C07243=1098.667,-38.202,448.879,175.841,14.477,151.943
C07244=1098.673,-37.951,448.867,175.843,14.477,151.943
C07245=1098.679,-37.701,448.855,175.845,14.478,151.943
C07246=1098.684,-37.452,448.843,175.847,14.478,151.942
C07247=1098.691,-37.202,448.831,175.849,14.479,151.942
C07248=1098.697,-36.953,448.818,175.851,14.480,151.942
C07249=1098.702,-36.703,448.806,175.852,14.481,151.942
C07250=1098.708,-36.453,448.793,175.854,14.481,151.941
C07251=1098.714,-36.204,448.781,175.856,14.482,151.941
C07252=1098.720,-35.955,448.769,175.858,14.482,151.941
C07253=1098.726,-35.705,448.757,175.859,14.483,151.940
C07254=1098.732,-35.455,448.744,175.861,14.483,151.940
C07255=1098.738,-35.205,448.731,175.863,14.484,151.940
C07256=1098.743,-34.956,448.719,175.865,14.485,151.940
C07257=1098.749,-34.706,448.707,175.867,14.486,151.939
C07258=1098.755,-34.456,448.695,175.869,14.486,151.939
C07259=1098.761,-34.207,448.683,175.871,14.487,151.939
C07260=1098.767,-33.957,448.670,175.873,14.487,151.938
C07261=1098.773,-33.707,448.657,175.875,14.488,151.938
C07262=1098.778,-33.458,448.645,175.877,14.489,151.938
C07263=1098.784,-33.208,448.633,175.879,14.490,151.938
C07264=1098.790,-32.959,448.620,175.880,14.490,151.937
C07265=1098.797,-32.692,448.607,175.883,14.491,151.937
C07266=1098.803,-32.424,448.593,175.885,14.492,151.937
C07267=1098.809,-32.158,448.581,175.887,14.493,151.936
C07268=1098.815,-31.891,448.567,175.889,14.494,151.936
C07269=1098.821,-31.641,448.554,175.891,14.494,151.936
C07270=1098.827,-31.391,448.542,175.893,14.495,151.935
C07271=1098.832,-31.142,448.529,175.895,14.495,151.935
C07272=1098.838,-30.892,448.517,175.897,14.496,151.935
C07273=1098.845,-30.642,448.505,175.899,14.497,151.935
C07274=1098.851,-30.392,448.492,175.901,14.497,151.934
C07275=1098.857,-30.142,448.480,175.903,14.498,151.934
C07276=1098.862,-29.893,448.468,175.905,14.499,151.934
C07277=1098.868,-29.644,448.454,175.907,14.499,151.933
C07278=1098.874,-29.394,448.442,175.908,14.500,151.933
C07279=1098.880,-29.144,448.429,175.911,14.500,151.933
C07280=1098.886,-28.894,448.417,175.912,14.501,151.932
C07281=1098.891,-28.645,448.405,175.914,14.502,151.932
C07282=1098.897,-28.395,448.392,175.916,14.503,151.932
C07283=1098.903,-28.146,448.379,175.918,14.503,151.932
C07284=1098.909,-27.896,448.366,175.920,14.504,151.931
C07285=1098.916,-27.647,448.354,175.922,14.504,151.931
C07286=1098.921,-27.397,448.342,175.924,14.505,151.931
C07287=1098.928,-27.148,448.329,175.926,14.506,151.930
C07288=1098.933,-26.898,448.316,175.928,14.507,151.930
C07289=1098.939,-26.648,448.304,175.930,14.507,151.930
C07290=1098.945,-26.398,448.291,175.932,14.508,151.930
C07291=1098.950,-26.149,448.278,175.934,14.509,151.929
C07292=1098.956,-25.900,448.265,175.936,14.509,151.929
C07293=1098.962,-25.650,448.252,175.937,14.510,151.929
C07294=1098.968,-25.400,448.240,175.939,14.511,151.928
C07295=1098.974,-25.150,448.227,175.942,14.511,151.928
C07296=1098.979,-24.902,448.214,175.943,14.512,151.928
C07297=1098.985,-24.652,448.202,175.945,14.513,151.928
C07298=1098.991,-24.402,448.189,175.947,14.513,151.927
C07299=1098.997,-24.152,448.176,175.949,14.514,151.927
C07300=1099.003,-23.902,448.163,175.951,14.515,151.927
C07301=1099.008,-23.652,448.150,175.953,14.515,151.926
C07302=1099.014,-23.404,448.138,175.956,14.517,151.926
C07303=1099.020,-23.154,448.125,175.958,14.517,151.926
C07304=1099.026,-22.904,448.112,175.960,14.518,151.926
C07305=1099.032,-22.655,448.099,175.961,14.519,151.925
C07306=1099.038,-22.405,448.087,175.964,14.519,151.925
C07307=1099.044,-22.155,448.074,175.965,14.520,151.925
C07308=1099.049,-21.906,448.061,175.967,14.521,151.924
C07309=1099.055,-21.656,448.048,175.969,14.521,151.924
C07310=1099.061,-21.406,448.035,175.971,14.522,151.924
C07311=1099.067,-21.157,448.022,175.973,14.522,151.923
C07312=1099.073,-20.907,448.010,175.975,14.523,151.923
C07313=1099.079,-20.658,447.996,175.977,14.524,151.923
C07314=1099.085,-20.408,447.984,175.979,14.525,151.923
C07315=1099.090,-20.158,447.971,175.981,14.525,151.922
C07316=1099.096,-19.909,447.957,175.983,14.526,151.922
C07317=1099.102,-19.659,447.945,175.985,14.527,151.922
C07318=1099.108,-19.410,447.932,175.987,14.527,151.921
C07319=1099.114,-19.160,447.919,175.989,14.528,151.921
C07320=1099.119,-18.911,447.905,175.991,14.528,151.921
C07321=1099.125,-18.661,447.893,175.993,14.529,151.920
C07322=1099.131,-18.412,447.880,175.995,14.530,151.920
C07323=1099.137,-18.162,447.867,175.997,14.531,151.920
C07324=1099.143,-17.912,447.855,175.999,14.531,151.919
C07325=1099.149,-17.662,447.841,176.001,14.532,151.919
C07326=1099.154,-17.412,447.828,176.003,14.533,151.919
C07327=1099.161,-17.163,447.815,176.005,14.534,151.919
C07328=1099.167,-16.914,447.802,176.007,14.534,151.918
C07329=1099.173,-16.646,447.789,176.009,14.535,151.918
C07330=1099.179,-16.378,447.774,176.011,14.536,151.918
C07331=1099.185,-16.110,447.760,176.014,14.536,151.917
C07332=1099.192,-15.842,447.746,176.016,14.537,151.917
C07333=1099.198,-15.593,447.733,176.018,14.538,151.917
C07334=1099.203,-15.343,447.720,176.020,14.538,151.916
C07335=1099.209,-15.094,447.706,176.022,14.539,151.916
C07336=1099.215,-14.844,447.694,176.024,14.540,151.916
C07337=1099.221,-14.594,447.680,176.025,14.541,151.916
C07338=1099.227,-14.344,447.667,176.028,14.541,151.915
C07339=1099.233,-14.095,447.654,176.030,14.542,151.915
C07340=1099.238,-13.845,447.640,176.031,14.542,151.915
C07341=1099.244,-13.595,447.628,176.034,14.544,151.914
C07342=1099.249,-13.347,447.614,176.036,14.544,151.914
C07343=1099.255,-13.097,447.602,176.038,14.545,151.914
C07344=1099.261,-12.847,447.588,176.040,14.546,151.913
C07345=1099.267,-12.598,447.574,176.042,14.546,151.913
C07346=1099.273,-12.348,447.562,176.044,14.547,151.913
C07347=1099.278,-12.098,447.548,176.046,14.547,151.912
C07348=1099.284,-11.849,447.535,176.048,14.548,151.912
C07349=1099.290,-11.599,447.522,176.050,14.549,151.912
C07350=1099.296,-11.350,447.508,176.052,14.549,151.912
C07351=1099.302,-11.100,447.495,176.054,14.550,151.911
C07352=1099.307,-10.850,447.482,176.056,14.551,151.911
C07353=1099.313,-10.601,447.469,176.058,14.552,151.911
C07354=1099.319,-10.351,447.455,176.060,14.552,151.910
C07355=1099.325,-10.101,447.442,176.062,14.553,151.910
C07356=1099.331,-9.852,447.429,176.064,14.554,151.910
C07357=1099.336,-9.603,447.415,176.066,14.554,151.909
C07358=1099.343,-9.353,447.402,176.068,14.555,151.909
C07359=1099.348,-9.103,447.389,176.070,14.556,151.909
C07360=1099.354,-8.854,447.375,176.072,14.556,151.908
C07361=1099.359,-8.604,447.362,176.074,14.557,151.908
C07362=1099.366,-8.355,447.348,176.077,14.558,151.908
C07363=1099.371,-8.105,447.335,176.079,14.559,151.908
C07364=1099.377,-7.856,447.322,176.081,14.559,151.907
C07365=1099.383,-7.606,447.308,176.083,14.560,151.907
C07366=1099.389,-7.357,447.295,176.085,14.561,151.907
C07367=1099.395,-7.106,447.282,176.087,14.561,151.906
C07368=1099.401,-6.857,447.268,176.089,14.562,151.906
C07369=1099.407,-6.607,447.255,176.091,14.563,151.906
C07370=1099.412,-6.358,447.241,176.093,14.563,151.905
C07371=1099.419,-6.109,447.228,176.095,14.564,151.905
C07372=1099.424,-5.859,447.214,176.097,14.565,151.905
C07373=1099.430,-5.609,447.201,176.100,14.565,151.904
C07374=1099.436,-5.360,447.187,176.101,14.566,151.904
C07375=1099.442,-5.110,447.174,176.104,14.566,151.904
C07376=1099.447,-4.861,447.160,176.105,14.567,151.903
C07377=1099.453,-4.611,447.147,176.107,14.568,151.903
C07378=1099.459,-4.362,447.133,176.110,14.568,151.903
C07379=1099.466,-4.112,447.119,176.111,14.569,151.902
C07380=1099.471,-3.862,447.106,176.114,14.570,151.902
C07381=1099.476,-3.612,447.092,176.116,14.571,151.902
C07382=1099.483,-3.363,447.079,176.118,14.571,151.901
C07383=1099.488,-3.113,447.065,176.120,14.572,151.901
C07384=1099.494,-2.864,447.052,176.122,14.572,151.901
C07385=1099.500,-2.614,447.038,176.124,14.573,151.901
C07386=1099.505,-2.365,447.024,176.126,14.574,151.900
C07387=1099.511,-2.115,447.010,176.128,14.574,151.900
C07388=1099.517,-1.866,446.997,176.131,14.576,151.900
C07389=1099.522,-1.616,446.983,176.133,14.576,151.899
C07390=1099.528,-1.367,446.969,176.135,14.577,151.899
C07391=1099.534,-1.118,446.956,176.137,14.577,151.899
C07392=1099.540,-0.867,446.942,176.139,14.578,151.898
C07393=1099.546,-0.597,446.927,176.141,14.578,151.898
C07394=1099.552,-0.328,446.912,176.143,14.580,151.898
C07395=1099.559,-0.059,446.898,176.146,14.580,151.897
C07396=1099.564,0.211,446.883,176.147,14.581,151.897
C07397=1099.571,0.461,446.869,176.150,14.582,151.897
C07398=1099.576,0.710,446.855,176.152,14.583,151.896
C07399=1099.581,0.960,446.842,176.154,14.583,151.896
C07400=1099.587,1.209,446.828,176.156,14.584,151.896
C07401=1099.593,1.459,446.814,176.158,14.584,151.895
C07402=1099.599,1.708,446.800,176.160,14.585,151.895
C07403=1099.604,1.957,446.786,176.162,14.585,151.895
C07404=1099.610,2.207,446.772,176.165,14.587,151.894
C07405=1099.616,2.457,446.758,176.167,14.588,151.894
C07406=1099.622,2.706,446.745,176.169,14.588,151.894
C07407=1099.628,2.956,446.731,176.171,14.589,151.893
C07408=1099.633,3.205,446.717,176.173,14.589,151.893
C07409=1099.639,3.455,446.703,176.175,14.590,151.893
C07410=1099.644,3.705,446.689,176.178,14.591,151.892
C07411=1099.651,3.955,446.676,176.180,14.591,151.892
C07412=1099.657,4.204,446.661,176.182,14.592,151.892
C07413=1099.662,4.453,446.647,176.184,14.592,151.891
C07414=1099.668,4.703,446.633,176.186,14.593,151.891
C07415=1099.673,4.952,446.619,176.188,14.594,151.891
C07416=1099.679,5.201,446.606,176.190,14.594,151.890
C07417=1099.685,5.452,446.592,176.192,14.596,151.890
C07418=1099.691,5.701,446.577,176.195,14.596,151.890
C07419=1099.697,5.950,446.563,176.196,14.597,151.889
C07420=1099.702,6.200,446.550,176.199,14.597,151.889
C07421=1099.708,6.450,446.535,176.201,14.598,151.889
C07422=1099.714,6.699,446.522,176.203,14.598,151.888
C07423=1099.720,6.948,446.507,176.205,14.599,151.888
C07424=1099.726,7.198,446.494,176.208,14.600,151.888
C07425=1099.731,7.448,446.480,176.209,14.601,151.887
C07426=1099.737,7.698,446.466,176.212,14.601,151.887
C07427=1099.743,7.947,446.451,176.214,14.602,151.887
C07428=1099.749,8.196,446.438,176.216,14.602,151.886
C07429=1099.755,8.446,446.424,176.218,14.603,151.886
C07430=1099.761,8.696,446.410,176.221,14.604,151.886
C07431=1099.767,8.945,446.395,176.222,14.604,151.885
C07432=1099.772,9.194,446.381,176.225,14.605,151.885
C07433=1099.778,9.444,446.367,176.226,14.605,151.885
C07434=1099.784,9.694,446.352,176.229,14.606,151.884
C07435=1099.789,9.943,446.338,176.231,14.607,151.884
C07436=1099.795,10.193,446.325,176.234,14.607,151.884
C07437=1099.802,10.442,446.310,176.235,14.608,151.883
C07438=1099.807,10.692,446.296,176.238,14.608,151.883
C07439=1099.813,10.941,446.283,176.239,14.609,151.883
C07440=1099.819,11.190,446.268,176.242,14.610,151.882
C07441=1099.825,11.441,446.254,176.244,14.611,151.882
C07442=1099.830,11.690,446.240,176.246,14.611,151.881
C07443=1099.836,11.939,446.225,176.248,14.612,151.881
C07444=1099.842,12.189,446.211,176.251,14.612,151.881
C07445=1099.848,12.438,446.196,176.253,14.613,151.880
C07446=1099.853,12.688,446.183,176.255,14.614,151.880
C07447=1099.859,12.938,446.168,176.258,14.614,151.880
C07448=1099.865,13.187,446.154,176.259,14.615,151.879
C07449=1099.871,13.437,446.140,176.262,14.615,151.879
C07450=1099.878,13.686,446.126,176.264,14.616,151.879
C07451=1099.883,13.936,446.112,176.266,14.617,151.878
C07452=1099.889,14.185,446.097,176.269,14.617,151.878
C07453=1099.895,14.435,446.083,176.271,14.618,151.878
C07454=1099.901,14.684,446.068,176.273,14.618,151.877
C07455=1099.906,14.934,446.054,176.275,14.619,151.877
C07456=1099.912,15.183,446.039,176.277,14.619,151.876
C07457=1099.918,15.455,446.024,176.280,14.620,151.876
C07458=1099.924,15.726,446.008,176.282,14.621,151.876
C07459=1099.931,15.998,445.992,176.285,14.622,151.875
C07460=1099.938,16.269,445.977,176.287,14.622,151.875
C07461=1099.942,16.519,445.962,176.289,14.623,151.875
C07462=1099.948,16.768,445.948,176.291,14.623,151.874
C07463=1099.954,17.018,445.933,176.294,14.624,151.874
C07464=1099.960,17.267,445.919,176.296,14.625,151.874
C07465=1099.965,17.517,445.905,176.298,14.625,151.873
C07466=1099.972,17.767,445.890,176.300,14.626,151.873
C07467=1099.977,18.016,445.876,176.303,14.627,151.872
C07468=1099.984,18.266,445.861,176.305,14.627,151.872
C07469=1099.989,18.515,445.846,176.307,14.628,151.872
C07470=1099.994,18.765,445.832,176.309,14.628,151.871
C07471=1100.001,19.014,445.817,176.311,14.629,151.871
C07472=1100.006,19.264,445.803,176.314,14.630,151.871
C07473=1100.012,19.513,445.789,176.316,14.630,151.870
C07474=1100.018,19.762,445.774,176.318,14.631,151.870
C07475=1100.023,20.012,445.759,176.320,14.632,151.869
C07476=1100.029,20.262,445.744,176.322,14.632,151.869
C07477=1100.035,20.511,445.730,176.325,14.633,151.869
C07478=1100.041,20.761,445.716,176.327,14.634,151.868
C07479=1100.047,21.010,445.701,176.329,14.634,151.868
C07480=1100.052,21.259,445.686,176.331,14.635,151.868
C07481=1100.058,21.510,445.672,176.334,14.636,151.867
C07482=1100.064,21.759,445.657,176.336,14.636,151.867
C07483=1100.070,22.008,445.642,176.338,14.637,151.867
C07484=1100.075,22.258,445.628,176.340,14.637,151.866
C07485=1100.081,22.507,445.613,176.342,14.638,151.866
C07486=1100.087,22.757,445.598,176.345,14.639,151.865
C07487=1100.092,23.006,445.583,176.347,14.639,151.865
C07488=1100.098,23.256,445.569,176.350,14.639,151.865
C07489=1100.104,23.505,445.554,176.351,14.640,151.864
C07490=1100.110,23.754,445.540,176.354,14.641,151.864
C07491=1100.116,24.004,445.524,176.357,14.641,151.863
C07492=1100.121,24.254,445.510,176.358,14.642,151.863
C07493=1100.127,24.503,445.495,176.361,14.642,151.863
C07494=1100.132,24.753,445.480,176.363,14.643,151.862
C07495=1100.138,25.002,445.465,176.365,14.644,151.862
C07496=1100.144,25.252,445.451,176.368,14.644,151.862
C07497=1100.149,25.501,445.436,176.370,14.645,151.861
C07498=1100.156,25.751,445.421,176.372,14.645,151.861
C07499=1100.162,26.000,445.407,176.375,14.646,151.861
C07500=1100.167,26.250,445.391,176.377,14.647,151.860
C07501=1100.173,26.499,445.376,176.379,14.647,151.860
C07502=1100.179,26.748,445.361,176.381,14.647,151.859
C07503=1100.184,26.998,445.347,176.384,14.649,151.859
C07504=1100.190,27.248,445.332,176.386,14.649,151.859
C07505=1100.196,27.497,445.317,176.388,14.649,151.858
C07506=1100.202,27.747,445.302,176.390,14.650,151.858
C07507=1100.208,27.996,445.287,176.393,14.650,151.857
C07508=1100.214,28.246,445.272,176.395,14.651,151.857
C07509=1100.219,28.495,445.257,176.398,14.652,151.857
C07510=1100.225,28.744,445.242,176.400,14.652,151.856
C07511=1100.231,28.994,445.227,176.403,14.653,151.856
C07512=1100.237,29.243,445.212,176.405,14.654,151.856
C07513=1100.242,29.493,445.198,176.407,14.654,151.855
C07514=1100.248,29.743,445.183,176.409,14.654,151.855
C07515=1100.253,29.992,445.168,176.412,14.655,151.854
C07516=1100.259,30.242,445.153,176.414,14.655,151.854
C07517=1100.265,30.491,445.137,176.416,14.656,151.854
C07518=1100.271,30.741,445.123,176.418,14.656,151.853
C07519=1100.276,30.990,445.107,176.421,14.657,151.853
C07520=1100.282,31.240,445.092,176.423,14.658,151.852
C07521=1100.288,31.512,445.075,176.425,14.658,151.852
C07522=1100.295,31.785,445.059,176.428,14.659,151.851
C07523=1100.301,32.058,445.043,176.431,14.659,151.851
C07524=1100.307,32.331,445.026,176.434,14.660,151.851
C07525=1100.313,32.581,445.011,176.436,14.660,151.850
C07526=1100.318,32.830,444.996,176.438,14.661,151.850
C07527=1100.325,33.080,444.981,176.440,14.662,151.849
C07528=1100.330,33.329,444.966,176.443,14.663,151.849
C07529=1100.336,33.579,444.951,176.445,14.663,151.849
C07530=1100.341,33.827,444.935,176.447,14.663,151.848
C07531=1100.348,34.077,444.920,176.450,14.664,151.848
C07532=1100.353,34.327,444.905,176.452,14.664,151.847
C07533=1100.358,34.576,444.889,176.455,14.665,151.847
C07534=1100.365,34.826,444.874,176.456,14.665,151.847
C07535=1100.370,35.075,444.859,176.459,14.666,151.846
C07536=1100.376,35.325,444.844,176.462,14.667,151.846
C07537=1100.382,35.575,444.829,176.464,14.667,151.845
C07538=1100.388,35.823,444.813,176.466,14.667,151.845
C07539=1100.394,36.073,444.798,176.469,14.668,151.844
C07540=1100.399,36.322,444.783,176.471,14.669,151.844
C07541=1100.405,36.572,444.768,176.473,14.669,151.844
C07542=1100.411,36.822,444.752,176.475,14.669,151.843
C07543=1100.417,37.071,444.738,176.478,14.670,151.843
C07544=1100.422,37.320,444.721,176.481,14.670,151.842
C07545=1100.428,37.570,444.706,176.483,14.671,151.842
C07546=1100.434,37.819,444.691,176.486,14.672,151.841
C07547=1100.440,38.069,444.676,176.488,14.672,151.841
C07548=1100.445,38.318,444.660,176.490,14.672,151.841
C07549=1100.451,38.568,444.645,176.492,14.673,151.840
C07550=1100.457,38.818,444.629,176.495,14.674,151.840
C07551=1100.462,39.067,444.614,176.497,14.674,151.840
C07552=1100.468,39.316,444.598,176.499,14.675,151.839
C07553=1100.474,39.565,444.583,176.502,14.676,151.839
C07554=1100.479,39.815,444.568,176.504,14.676,151.838
C07555=1100.485,40.065,444.552,176.507,14.676,151.838
C07556=1100.490,40.314,444.536,176.509,14.676,151.837
C07557=1100.497,40.563,444.521,176.512,14.677,151.837
C07558=1100.502,40.813,444.506,176.514,14.678,151.837
C07559=1100.508,41.062,444.490,176.516,14.678,151.836
C07560=1100.513,41.312,444.474,176.519,14.679,151.836
C07561=1100.519,41.562,444.459,176.521,14.679,151.835
C07562=1100.525,41.810,444.444,176.524,14.680,151.835
C07563=1100.531,42.060,444.428,176.526,14.680,151.834
C07564=1100.536,42.310,444.413,176.529,14.681,151.834
C07565=1100.542,42.559,444.397,176.531,14.681,151.834
C07566=1100.548,42.809,444.382,176.533,14.681,151.833
C07567=1100.554,43.058,444.365,176.536,14.682,151.833
C07568=1100.559,43.307,444.350,176.538,14.683,151.832
C07569=1100.565,43.557,444.335,176.541,14.683,151.832
C07570=1100.571,43.806,444.318,176.544,14.684,151.831
C07571=1100.576,44.056,444.303,176.546,14.684,151.831
C07572=1100.582,44.305,444.287,176.548,14.684,151.830
C07573=1100.587,44.555,444.271,176.550,14.684,151.830
C07574=1100.592,44.804,444.256,176.553,14.685,151.830
C07575=1100.599,45.053,444.241,176.555,14.686,151.829
C07576=1100.605,45.303,444.225,176.558,14.686,151.829
C07577=1100.610,45.552,444.209,176.561,14.687,151.828
C07578=1100.616,45.802,444.194,176.563,14.687,151.828
C07579=1100.622,46.051,444.177,176.565,14.688,151.827
C07580=1100.627,46.301,444.162,176.568,14.689,151.827
C07581=1100.633,46.550,444.146,176.570,14.689,151.827
C07582=1100.638,46.800,444.130,176.572,14.689,151.826
C07583=1100.644,47.049,444.114,176.575,14.690,151.826
C07584=1100.649,47.298,444.099,176.577,14.690,151.825
C07585=1100.656,47.572,444.081,176.580,14.691,151.825
C07586=1100.662,47.845,444.064,176.583,14.691,151.824
C07587=1100.668,48.117,444.047,176.586,14.692,151.824
C07588=1100.674,48.391,444.029,176.588,14.692,151.823
C07589=1100.680,48.640,444.013,176.591,14.692,151.823
C07590=1100.685,48.889,443.997,176.594,14.693,151.822
C07591=1100.691,49.139,443.982,176.596,14.694,151.822
C07592=1100.697,49.388,443.965,176.598,14.694,151.822
C07593=1100.702,49.637,443.950,176.601,14.695,151.821
C07594=1100.708,49.887,443.934,176.603,14.695,151.821
C07595=1100.714,50.136,443.918,176.605,14.695,151.820
C07596=1100.720,50.386,443.902,176.609,14.696,151.820
C07597=1100.726,50.636,443.886,176.611,14.696,151.819
C07598=1100.731,50.884,443.870,176.613,14.697,151.819
C07599=1100.737,51.134,443.854,176.616,14.698,151.818
C07600=1100.743,51.383,443.838,176.618,14.698,151.818
C07601=1100.748,51.633,443.821,176.621,14.698,151.817
C07602=1100.753,51.883,443.806,176.624,14.699,151.817
C07603=1100.759,52.132,443.790,176.626,14.699,151.817
C07604=1100.765,52.381,443.774,176.628,14.699,151.816
C07605=1100.770,52.631,443.758,176.631,14.700,151.815
C07606=1100.776,52.880,443.742,176.633,14.700,151.815
C07607=1100.782,53.130,443.726,176.636,14.700,151.815
C07608=1100.788,53.378,443.710,176.638,14.701,151.814
C07609=1100.793,53.628,443.694,176.641,14.701,151.814
C07610=1100.799,53.878,443.678,176.643,14.702,151.813
C07611=1100.805,54.127,443.662,176.645,14.702,151.813
C07612=1100.811,54.376,443.645,176.648,14.703,151.812
C07613=1100.816,54.627,443.629,176.651,14.703,151.812
C07614=1100.822,54.876,443.613,176.653,14.703,151.811
C07615=1100.827,55.125,443.597,176.656,14.704,151.811
C07616=1100.833,55.374,443.581,176.659,14.704,151.810
C07617=1100.839,55.623,443.565,176.661,14.704,151.810
C07618=1100.845,55.873,443.548,176.664,14.705,151.809
C07619=1100.851,56.123,443.533,176.666,14.705,151.809
C07620=1100.856,56.372,443.516,176.668,14.705,151.808
C07621=1100.862,56.622,443.500,176.671,14.706,151.808
C07622=1100.868,56.871,443.483,176.674,14.706,151.807
C07623=1100.874,57.120,443.467,176.676,14.706,151.807
C07624=1100.879,57.369,443.451,176.679,14.707,151.806
C07625=1100.885,57.618,443.435,176.681,14.707,151.806
C07626=1100.891,57.868,443.419,176.684,14.707,151.806
C07627=1100.896,58.118,443.403,176.687,14.708,151.805
C07628=1100.902,58.367,443.386,176.689,14.708,151.805
C07629=1100.908,58.617,443.370,176.692,14.708,151.804
C07630=1100.914,58.866,443.354,176.695,14.709,151.804
C07631=1100.920,59.115,443.338,176.697,14.709,151.803
C07632=1100.925,59.365,443.321,176.700,14.710,151.803
C07633=1100.931,59.614,443.305,176.702,14.710,151.802
C07634=1100.937,59.864,443.288,176.705,14.710,151.802
C07635=1100.943,60.113,443.272,176.708,14.711,151.801
C07636=1100.949,60.362,443.256,176.710,14.711,151.801
C07637=1100.954,60.612,443.239,176.712,14.711,151.800
C07638=1100.960,60.861,443.223,176.716,14.712,151.799
C07639=1100.966,61.111,443.206,176.718,14.712,151.799
C07640=1100.972,61.360,443.190,176.720,14.712,151.798
C07641=1100.977,61.610,443.173,176.723,14.713,151.798
C07642=1100.983,61.859,443.157,176.726,14.713,151.797
C07643=1100.989,62.109,443.141,176.728,14.713,151.797
C07644=1100.995,62.357,443.124,176.731,14.714,151.796
C07645=1101.001,62.607,443.107,176.734,14.714,151.796
C07646=1101.006,62.856,443.091,176.736,14.714,151.795
C07647=1101.012,63.106,443.074,176.739,14.715,151.795
C07648=1101.018,63.355,443.058,176.741,14.715,151.794
C07649=1101.025,63.627,443.040,176.745,14.715,151.794
C07650=1101.030,63.901,443.022,176.747,14.715,151.793
C07651=1101.037,64.174,443.004,176.750,14.716,151.793
C07652=1101.043,64.446,442.986,176.753,14.716,151.792
C07653=1101.049,64.695,442.970,176.756,14.716,151.792
C07654=1101.055,64.945,442.953,176.758,14.717,151.791
C07655=1101.061,65.194,442.936,176.761,14.716,151.791
C07656=1101.066,65.443,442.919,176.764,14.717,151.790
C07657=1101.072,65.693,442.903,176.766,14.717,151.790
C07658=1101.078,65.942,442.886,176.769,14.717,151.789
C07659=1101.083,66.192,442.870,176.772,14.718,151.789
C07660=1101.089,66.441,442.853,176.774,14.718,151.788
C07661=1101.095,66.690,442.836,176.776,14.718,151.788
C07662=1101.101,66.939,442.819,176.780,14.719,151.787
C07663=1101.106,67.189,442.803,176.782,14.719,151.786
C07664=1101.112,67.438,442.786,176.785,14.720,151.786
C07665=1101.117,67.688,442.769,176.788,14.719,151.785
C07666=1101.124,67.937,442.752,176.790,14.720,151.785
C07667=1101.129,68.187,442.735,176.793,14.720,151.784
C07668=1101.135,68.436,442.719,176.796,14.720,151.784
C07669=1101.141,68.686,442.701,176.798,14.720,151.783
C07670=1101.146,68.935,442.685,176.801,14.721,151.783
C07671=1101.152,69.185,442.668,176.804,14.721,151.782
C07672=1101.158,69.433,442.651,176.806,14.722,151.782
C07673=1101.163,69.683,442.635,176.809,14.722,151.781
C07674=1101.169,69.932,442.618,176.812,14.721,151.781
C07675=1101.174,70.182,442.601,176.814,14.722,151.780
C07676=1101.181,70.431,442.584,176.817,14.722,151.780
C07677=1101.186,70.680,442.568,176.819,14.722,151.779
C07678=1101.191,70.929,442.550,176.822,14.723,151.779
C07679=1101.197,71.179,442.534,176.825,14.723,151.778
C07680=1101.203,71.429,442.517,176.828,14.724,151.777
C07681=1101.209,71.678,442.500,176.830,14.724,151.777
C07682=1101.215,71.927,442.483,176.833,14.724,151.776
C07683=1101.220,72.176,442.465,176.836,14.724,151.776
C07684=1101.226,72.426,442.449,176.838,14.725,151.775
C07685=1101.231,72.675,442.432,176.841,14.724,151.775
C07686=1101.237,72.925,442.414,176.844,14.725,151.774
C07687=1101.243,73.174,442.398,176.847,14.725,151.774
C07688=1101.248,73.423,442.381,176.850,14.726,151.773
C07689=1101.255,73.673,442.364,176.852,14.726,151.773
C07690=1101.260,73.922,442.346,176.855,14.725,151.772
C07691=1101.265,74.172,442.330,176.858,14.726,151.771
C07692=1101.272,74.420,442.313,176.860,14.726,151.771
C07693=1101.277,74.670,442.296,176.863,14.726,151.770
C07694=1101.282,74.919,442.278,176.866,14.727,151.770
C07695=1101.288,75.169,442.261,176.868,14.727,151.769
C07696=1101.295,75.418,442.244,176.872,14.727,151.769
C07697=1101.300,75.668,442.227,176.874,14.727,151.768
C07698=1101.305,75.917,442.210,176.876,14.727,151.768
C07699=1101.311,76.166,442.193,176.880,14.728,151.767
C07700=1101.317,76.415,442.176,176.882,14.728,151.766
C07701=1101.322,76.665,442.159,176.885,14.728,151.766
C07702=1101.329,76.914,442.142,176.888,14.728,151.765
C07703=1101.334,77.163,442.124,176.890,14.728,151.765
C07704=1101.340,77.413,442.107,176.893,14.729,151.764
C07705=1101.345,77.662,442.090,176.896,14.729,151.764
C07706=1101.351,77.911,442.073,176.898,14.729,151.763
C07707=1101.357,78.161,442.055,176.902,14.729,151.762
C07708=1101.363,78.410,442.038,176.904,14.729,151.762
C07709=1101.368,78.660,442.021,176.907,14.730,151.761
C07710=1101.373,78.909,442.003,176.910,14.729,151.761
C07711=1101.380,79.158,441.986,176.912,14.729,151.760
C07712=1101.385,79.408,441.969,176.916,14.730,151.760
C07713=1101.391,79.680,441.950,176.918,14.730,151.759
C07714=1101.397,79.953,441.931,176.922,14.730,151.758
C07715=1101.404,80.226,441.911,176.925,14.731,151.758
C07716=1101.410,80.499,441.893,176.927,14.731,151.757
C07717=1101.416,80.747,441.876,176.931,14.731,151.757
C07718=1101.421,80.997,441.859,176.933,14.731,151.756
C07719=1101.427,81.246,441.841,176.936,14.731,151.755
C07720=1101.432,81.495,441.824,176.939,14.731,151.755
C07721=1101.438,81.745,441.806,176.941,14.731,151.754
C07722=1101.444,81.995,441.789,176.945,14.732,151.754
C07723=1101.449,82.244,441.771,176.947,14.732,151.753
C07724=1101.455,82.493,441.754,176.950,14.732,151.752
C07725=1101.461,82.742,441.736,176.953,14.732,151.752
C07726=1101.466,82.991,441.718,176.955,14.732,151.751
C07727=1101.472,83.241,441.701,176.959,14.732,151.751
C07728=1101.477,83.490,441.684,176.961,14.732,151.750
C07729=1101.483,83.740,441.666,176.965,14.733,151.750
C07730=1101.489,83.989,441.648,176.967,14.733,151.749
C07731=1101.494,84.238,441.631,176.970,14.733,151.748
C07732=1101.500,84.488,441.613,176.973,14.733,151.748
C07733=1101.506,84.737,441.597,176.975,14.733,151.747
C07734=1101.512,84.986,441.579,176.979,14.733,151.747
C07735=1101.517,85.235,441.561,176.981,14.733,151.746
C07736=1101.523,85.485,441.543,176.984,14.733,151.745
C07737=1101.529,85.734,441.526,176.987,14.734,151.745
C07738=1101.534,85.983,441.508,176.989,14.734,151.744
C07739=1101.541,86.233,441.490,176.993,14.734,151.744
C07740=1101.546,86.482,441.473,176.995,14.734,151.743
C07741=1101.552,86.731,441.455,176.998,14.733,151.742
C07742=1101.558,86.980,441.437,177.001,14.734,151.742
C07743=1101.563,87.230,441.420,177.004,14.734,151.741
C07744=1101.569,87.479,441.402,177.007,14.734,151.741
C07745=1101.575,87.728,441.384,177.010,14.734,151.740
C07746=1101.580,87.978,441.366,177.012,14.734,151.739
C07747=1101.586,88.227,441.348,177.016,14.734,151.739
C07748=1101.591,88.476,441.331,177.018,14.734,151.738
C07749=1101.597,88.725,441.313,177.021,14.735,151.737
C07750=1101.603,88.975,441.295,177.024,14.734,151.737
C07751=1101.608,89.224,441.278,177.026,14.734,151.736
C07752=1101.615,89.474,441.260,177.030,14.734,151.736
C07753=1101.620,89.723,441.242,177.033,14.734,151.735
C07754=1101.626,89.972,441.224,177.036,14.735,151.734
C07755=1101.632,90.222,441.207,177.038,14.735,151.734
C07756=1101.637,90.471,441.189,177.042,14.735,151.733
C07757=1101.643,90.721,441.171,177.044,14.735,151.732
C07758=1101.649,90.970,441.153,177.047,14.735,151.732
C07759=1101.655,91.218,441.135,177.050,14.735,151.731
C07760=1101.660,91.468,441.117,177.053,14.734,151.731
C07761=1101.666,91.717,441.099,177.056,14.735,151.730
C07762=1101.672,91.967,441.081,177.059,14.735,151.729
C07763=1101.677,92.216,441.064,177.061,14.735,151.729
C07764=1101.682,92.465,441.045,177.065,14.735,151.728
C07765=1101.688,92.715,441.027,177.067,14.735,151.727
C07766=1101.694,92.963,441.009,177.071,14.735,151.727
C07767=1101.700,93.213,440.991,177.073,14.735,151.726
C07768=1101.706,93.462,440.974,177.077,14.735,151.726
C07769=1101.710,93.712,440.956,177.079,14.735,151.725
C07770=1101.717,93.961,440.938,177.082,14.735,151.724
C07771=1101.722,94.210,440.919,177.085,14.736,151.724
C07772=1101.728,94.460,440.901,177.088,14.735,151.723
C07773=1101.733,94.709,440.883,177.091,14.736,151.722
C07774=1101.739,94.959,440.865,177.094,14.735,151.722
C07775=1101.745,95.207,440.847,177.097,14.735,151.721
C07776=1101.750,95.456,440.829,177.100,14.735,151.721
C07777=1101.757,95.730,440.809,177.103,14.735,151.720
C07778=1101.763,96.002,440.789,177.106,14.735,151.719
C07779=1101.769,96.275,440.769,177.109,14.735,151.718
C07780=1101.775,96.547,440.749,177.113,14.735,151.718
C07781=1101.781,96.797,440.732,177.116,14.735,151.717
C07782=1101.787,97.046,440.713,177.118,14.735,151.716
C07783=1101.792,97.295,440.695,177.122,14.735,151.716
C07784=1101.798,97.545,440.677,177.124,14.735,151.715
C07785=1101.803,97.793,440.658,177.128,14.735,151.714
C07786=1101.809,98.043,440.640,177.130,14.735,151.714
C07787=1101.815,98.292,440.623,177.134,14.735,151.713
C07788=1101.821,98.542,440.603,177.136,14.735,151.712
C07789=1101.826,98.791,440.586,177.140,14.735,151.712
C07790=1101.833,99.040,440.567,177.142,14.735,151.711
C07791=1101.837,99.289,440.549,177.145,14.735,151.710
C07792=1101.844,99.539,440.531,177.149,14.735,151.710
C07793=1101.850,99.788,440.512,177.151,14.735,151.709
C07794=1101.855,100.037,440.494,177.155,14.735,151.708
C07795=1101.861,100.287,440.476,177.157,14.735,151.708
C07796=1101.867,100.536,440.458,177.161,14.735,151.707
C07797=1101.872,100.785,440.439,177.164,14.734,151.706
C07798=1101.878,101.034,440.421,177.166,14.734,151.706
C07799=1101.884,101.283,440.402,177.170,14.734,151.705
C07800=1101.889,101.533,440.384,177.172,14.734,151.704
C07801=1101.895,101.782,440.365,177.176,14.734,151.704
C07802=1101.901,102.032,440.347,177.179,14.734,151.703
C07803=1101.906,102.280,440.328,177.182,14.734,151.702
C07804=1101.912,102.530,440.310,177.185,14.734,151.702
C07805=1101.917,102.779,440.292,177.187,14.734,151.701
C07806=1101.924,103.028,440.273,177.191,14.734,151.700
C07807=1101.928,103.277,440.255,177.193,14.734,151.700
C07808=1101.935,103.526,440.236,177.197,14.734,151.699
C07809=1101.940,103.776,440.218,177.200,14.733,151.698
C07810=1101.945,104.025,440.199,177.203,14.734,151.698
C07811=1101.951,104.275,440.181,177.206,14.733,151.697
C07812=1101.957,104.524,440.162,177.209,14.734,151.696
C07813=1101.963,104.773,440.143,177.212,14.733,151.696
C07814=1101.968,105.022,440.125,177.215,14.733,151.695
C07815=1101.974,105.271,440.106,177.218,14.733,151.694
C07816=1101.980,105.521,440.087,177.221,14.733,151.693
C07817=1101.985,105.770,440.069,177.224,14.733,151.693
C07818=1101.991,106.019,440.050,177.227,14.733,151.692
C07819=1101.997,106.269,440.031,177.231,14.733,151.691
C07820=1102.002,106.518,440.014,177.233,14.732,151.691
C07821=1102.008,106.767,439.994,177.237,14.733,151.690
C07822=1102.013,107.016,439.976,177.239,14.732,151.689
C07823=1102.019,107.265,439.957,177.243,14.732,151.689
C07824=1102.025,107.515,439.938,177.246,14.732,151.688
C07825=1102.031,107.763,439.920,177.248,14.732,151.687
C07826=1102.036,108.013,439.901,177.252,14.732,151.686
C07827=1102.042,108.262,439.882,177.255,14.731,151.686
C07828=1102.048,108.511,439.864,177.258,14.732,151.685
C07829=1102.053,108.761,439.845,177.261,14.731,151.684
C07830=1102.059,109.010,439.826,177.264,14.731,151.684
C07831=1102.065,109.259,439.807,177.267,14.731,151.683
C07832=1102.070,109.508,439.788,177.271,14.731,151.682
C07833=1102.076,109.758,439.769,177.273,14.731,151.682
C07834=1102.082,110.007,439.751,177.276,14.730,151.681
C07835=1102.087,110.256,439.732,177.280,14.730,151.680
C07836=1102.093,110.505,439.713,177.283,14.730,151.679
C07837=1102.099,110.755,439.694,177.286,14.730,151.679
C07838=1102.105,111.004,439.675,177.289,14.729,151.678
C07839=1102.110,111.253,439.656,177.292,14.730,151.677
C07840=1102.117,111.502,439.637,177.295,14.729,151.676
C07841=1102.122,111.775,439.617,177.299,14.729,151.676
C07842=1102.129,112.048,439.596,177.303,14.729,151.675
C07843=1102.135,112.320,439.576,177.305,14.729,151.674
C07844=1102.141,112.593,439.554,177.309,14.729,151.673
C07845=1102.147,112.843,439.535,177.312,14.728,151.673
C07846=1102.152,113.092,439.516,177.315,14.728,151.672
C07847=1102.158,113.341,439.497,177.318,14.728,151.671
C07848=1102.164,113.590,439.478,177.322,14.728,151.670
C07849=1102.170,113.840,439.459,177.325,14.727,151.670
C07850=1102.175,114.088,439.440,177.328,14.727,151.669
C07851=1102.180,114.338,439.421,177.331,14.727,151.668
C07852=1102.187,114.587,439.402,177.334,14.727,151.667
C07853=1102.193,114.836,439.383,177.337,14.727,151.667
C07854=1102.198,115.085,439.364,177.341,14.727,151.666
C07855=1102.203,115.334,439.345,177.344,14.726,151.665
C07856=1102.209,115.584,439.326,177.346,14.726,151.664
C07857=1102.214,115.833,439.307,177.350,14.726,151.664
C07858=1102.220,116.082,439.287,177.353,14.725,151.663
C07859=1102.225,116.331,439.268,177.356,14.725,151.662
C07860=1102.231,116.581,439.249,177.359,14.725,151.661
C07861=1102.237,116.829,439.229,177.363,14.725,151.661
C07862=1102.242,117.078,439.210,177.366,14.724,151.660
C07863=1102.248,117.328,439.191,177.369,14.725,151.659
C07864=1102.254,117.577,439.172,177.372,14.724,151.659
C07865=1102.259,117.827,439.152,177.376,14.724,151.658
C07866=1102.264,118.075,439.134,177.378,14.724,151.657
C07867=1102.270,118.325,439.114,177.382,14.724,151.656
C07868=1102.276,118.574,439.095,177.385,14.723,151.656
C07869=1102.282,118.823,439.075,177.389,14.723,151.655
C07870=1102.287,119.073,439.056,177.391,14.723,151.654
C07871=1102.293,119.321,439.037,177.395,14.723,151.653
C07872=1102.298,119.571,439.018,177.398,14.722,151.653
C07873=1102.304,119.820,438.998,177.401,14.722,151.652
C07874=1102.310,120.069,438.979,177.404,14.722,151.651
C07875=1102.316,120.318,438.959,177.407,14.721,151.650
C07876=1102.321,120.568,438.940,177.411,14.722,151.650
C07877=1102.327,120.816,438.920,177.413,14.721,151.649
C07878=1102.332,121.066,438.901,177.417,14.721,151.648
C07879=1102.337,121.315,438.881,177.420,14.721,151.647
C07880=1102.343,121.565,438.862,177.423,14.721,151.647
C07881=1102.349,121.813,438.842,177.427,14.720,151.646
C07882=1102.355,122.063,438.823,177.430,14.720,151.645
C07883=1102.360,122.312,438.804,177.433,14.719,151.644
C07884=1102.366,122.560,438.784,177.437,14.719,151.643
C07885=1102.371,122.810,438.765,177.439,14.719,151.643
C07886=1102.377,123.059,438.746,177.443,14.719,151.642
C07887=1102.383,123.308,438.726,177.446,14.718,151.641
C07888=1102.389,123.557,438.706,177.450,14.718,151.640
C07889=1102.394,123.807,438.686,177.453,14.718,151.639
C07890=1102.400,124.056,438.667,177.456,14.718,151.639
C07891=1102.405,124.305,438.647,177.459,14.717,151.638
C07892=1102.411,124.554,438.627,177.462,14.716,151.637
C07893=1102.417,124.804,438.608,177.466,14.716,151.636
C07894=1102.423,125.053,438.588,177.469,14.716,151.636
C07895=1102.429,125.302,438.569,177.472,14.715,151.635
C07896=1102.434,125.551,438.548,177.475,14.715,151.634
C07897=1102.440,125.801,438.529,177.479,14.715,151.633
C07898=1102.446,126.049,438.509,177.482,14.714,151.632
C07899=1102.451,126.299,438.490,177.486,14.714,151.632
C07900=1102.457,126.547,438.470,177.488,14.714,151.631
C07901=1102.463,126.796,438.451,177.492,14.713,151.630
C07902=1102.468,127.045,438.431,177.495,14.713,151.629
C07903=1102.473,127.295,438.411,177.499,14.713,151.628
C07904=1102.479,127.544,438.391,177.502,14.712,151.627
C07905=1102.486,127.817,438.370,177.505,14.712,151.627
C07906=1102.492,128.090,438.348,177.509,14.712,151.626
C07907=1102.499,128.362,438.326,177.513,14.711,151.625
C07908=1102.505,128.635,438.305,177.516,14.711,151.624
C07909=1102.511,128.885,438.286,177.519,14.710,151.623
C07910=1102.516,129.134,438.265,177.523,14.710,151.622
C07911=1102.522,129.382,438.245,177.526,14.709,151.622
C07912=1102.528,129.632,438.226,177.530,14.709,151.621
C07913=1102.534,129.881,438.206,177.533,14.708,151.620
C07914=1102.539,130.130,438.185,177.537,14.708,151.619
C07915=1102.545,130.379,438.166,177.539,14.707,151.618
C07916=1102.551,130.628,438.146,177.543,14.707,151.617
C07917=1102.557,130.877,438.126,177.546,14.707,151.617
C07918=1102.562,131.127,438.106,177.550,14.706,151.616
C07919=1102.568,131.375,438.086,177.553,14.706,151.615
C07920=1102.574,131.624,438.066,177.557,14.705,151.614
C07921=1102.580,131.873,438.046,177.560,14.705,151.613
C07922=1102.585,132.124,438.026,177.564,14.705,151.612
C07923=1102.591,132.372,438.006,177.566,14.704,151.612
C07924=1102.597,132.621,437.986,177.570,14.704,151.611
C07925=1102.603,132.870,437.966,177.573,14.703,151.610
C07926=1102.608,133.120,437.947,177.577,14.703,151.609
C07927=1102.613,133.369,437.926,177.580,14.702,151.608
C07928=1102.619,133.618,437.906,177.584,14.702,151.607
C07929=1102.625,133.867,437.885,177.587,14.702,151.607
C07930=1102.631,134.116,437.865,177.591,14.701,151.606
C07931=1102.636,134.365,437.846,177.593,14.701,151.605
C07932=1102.642,134.614,437.826,177.597,14.701,151.604
C07933=1102.647,134.863,437.805,177.600,14.700,151.603
C07934=1102.653,135.112,437.785,177.604,14.700,151.602
C07935=1102.659,135.362,437.765,177.607,14.699,151.602
C07936=1102.665,135.611,437.744,177.611,14.699,151.601
C07937=1102.670,135.860,437.725,177.614,14.698,151.600
C07938=1102.676,136.109,437.705,177.617,14.698,151.599
C07939=1102.682,136.358,437.685,177.621,14.697,151.598
C07940=1102.687,136.607,437.664,177.624,14.697,151.597
C07941=1102.693,136.856,437.644,177.627,14.696,151.597
C07942=1102.698,137.105,437.623,177.631,14.696,151.596
C07943=1102.705,137.355,437.603,177.634,14.695,151.595
C07944=1102.710,137.604,437.583,177.638,14.695,151.594
C07945=1102.715,137.853,437.562,177.641,14.694,151.593
C07946=1102.721,138.102,437.542,177.644,14.693,151.592
C07947=1102.727,138.351,437.522,177.648,14.693,151.591
C07948=1102.733,138.600,437.502,177.651,14.692,151.591
C07949=1102.738,138.849,437.481,177.655,14.692,151.590
C07950=1102.744,139.098,437.461,177.658,14.692,151.589
C07951=1102.750,139.347,437.440,177.662,14.691,151.588
C07952=1102.755,139.597,437.420,177.665,14.690,151.587
C07953=1102.761,139.845,437.400,177.669,14.690,151.586
C07954=1102.766,140.094,437.379,177.672,14.690,151.585
C07955=1102.773,140.344,437.359,177.675,14.689,151.585
C07956=1102.778,140.593,437.338,177.679,14.688,151.584
C07957=1102.783,140.842,437.318,177.682,14.688,151.583
C07958=1102.789,141.091,437.298,177.685,14.688,151.582
C07959=1102.795,141.340,437.276,177.689,14.687,151.581
C07960=1102.801,141.589,437.255,177.692,14.686,151.580
C07961=1102.807,141.838,437.236,177.696,14.686,151.579
C07962=1102.812,142.087,437.215,177.699,14.686,151.578
C07963=1102.817,142.336,437.194,177.703,14.685,151.578
C07964=1102.822,142.586,437.174,177.706,14.684,151.577
C07965=1102.829,142.835,437.154,177.710,14.684,151.576
C07966=1102.835,143.084,437.132,177.713,14.684,151.575
C07967=1102.840,143.333,437.112,177.717,14.683,151.574
C07968=1102.846,143.582,437.092,177.720,14.682,151.573
C07969=1102.852,143.854,437.069,177.724,14.682,151.572
C07970=1102.858,144.127,437.047,177.728,14.681,151.571
C07971=1102.864,144.399,437.024,177.732,14.681,151.570
C07972=1102.870,144.672,437.001,177.735,14.680,151.569
C07973=1102.877,144.921,436.980,177.739,14.680,151.568
C07974=1102.882,145.170,436.959,177.742,14.679,151.568
C07975=1102.888,145.419,436.939,177.746,14.679,151.567
C07976=1102.893,145.668,436.919,177.749,14.678,151.566
C07977=1102.899,145.917,436.897,177.753,14.677,151.565
C07978=1102.904,146.167,436.876,177.756,14.676,151.564
C07979=1102.910,146.416,436.856,177.760,14.676,151.563
C07980=1102.917,146.665,436.835,177.763,14.675,151.562
C07981=1102.922,146.914,436.814,177.767,14.675,151.561
C07982=1102.927,147.163,436.794,177.770,14.674,151.560
C07983=1102.933,147.412,436.772,177.774,14.674,151.559
C07984=1102.939,147.661,436.752,177.777,14.673,151.558
C07985=1102.945,147.909,436.731,177.781,14.672,151.558
C07986=1102.951,148.159,436.710,177.785,14.671,151.557
C07987=1102.956,148.408,436.689,177.788,14.671,151.556
C07988=1102.961,148.657,436.668,177.792,14.671,151.555
C07989=1102.967,148.907,436.647,177.795,14.670,151.554
C07990=1102.973,149.155,436.626,177.799,14.670,151.553
C07991=1102.978,149.404,436.605,177.803,14.669,151.552
C07992=1102.984,149.653,436.584,177.806,14.669,151.551
C07993=1102.990,149.903,436.563,177.810,14.668,151.550
C07994=1102.995,150.151,436.542,177.813,14.667,151.549
C07995=1103.001,150.401,436.521,177.817,14.666,151.548
C07996=1103.007,150.649,436.500,177.821,14.666,151.548
C07997=1103.013,150.898,436.480,177.824,14.665,151.547
C07998=1103.019,151.147,436.458,177.828,14.665,151.546
C07999=1103.024,151.397,436.438,177.831,14.664,151.545
C08000=1103.030,151.646,436.416,177.835,14.664,151.544
C08001=1103.035,151.895,436.395,177.838,14.663,151.543
C08002=1103.041,152.143,436.374,177.842,14.662,151.542
C08003=1103.047,152.393,436.353,177.845,14.661,151.541
C08004=1103.052,152.642,436.332,177.849,14.661,151.540
C08005=1103.059,152.891,436.310,177.852,14.660,151.539
C08006=1103.063,153.140,436.289,177.856,14.660,151.538
C08007=1103.069,153.389,436.268,177.859,14.659,151.537
C08008=1103.075,153.638,436.246,177.863,14.658,151.537
C08009=1103.080,153.887,436.226,177.866,14.658,151.536
C08010=1103.086,154.136,436.204,177.871,14.657,151.535
C08011=1103.092,154.385,436.183,177.874,14.656,151.534
C08012=1103.097,154.634,436.162,177.878,14.656,151.533
C08013=1103.103,154.883,436.141,177.881,14.655,151.532
C08014=1103.109,155.132,436.119,177.885,14.654,151.531
C08015=1103.115,155.382,436.098,177.888,14.653,151.530
C08016=1103.120,155.630,436.077,177.892,14.653,151.529
C08017=1103.126,155.879,436.055,177.895,14.652,151.528
C08018=1103.132,156.128,436.035,177.899,14.652,151.527
C08019=1103.137,156.378,436.013,177.903,14.650,151.526
C08020=1103.143,156.626,435.991,177.906,14.650,151.525
C08021=1103.149,156.876,435.970,177.910,14.649,151.524
C08022=1103.154,157.124,435.949,177.914,14.649,151.523
C08023=1103.160,157.374,435.928,177.918,14.648,151.522
C08024=1103.166,157.622,435.906,177.921,14.647,151.521
C08025=1103.171,157.871,435.884,177.925,14.647,151.520
C08026=1103.177,158.120,435.863,177.928,14.646,151.520
C08027=1103.182,158.369,435.842,177.932,14.645,151.518
C08028=1103.188,158.619,435.821,177.935,14.644,151.518
C08029=1103.194,158.868,435.799,177.939,14.644,151.517
C08030=1103.199,159.117,435.777,177.943,14.643,151.516
C08031=1103.205,159.366,435.756,177.947,14.643,151.515
C08032=1103.211,159.615,435.734,177.950,14.642,151.514
C08033=1103.217,159.887,435.711,177.954,14.641,151.513
C08034=1103.223,160.159,435.687,177.958,14.640,151.512
C08035=1103.230,160.432,435.663,177.962,14.639,151.511
C08036=1103.236,160.704,435.640,177.966,14.638,151.509
C08037=1103.241,160.952,435.618,177.970,14.638,151.509
C08038=1103.247,161.202,435.596,177.973,14.637,151.508
C08039=1103.253,161.450,435.575,177.977,14.636,151.507
C08040=1103.258,161.700,435.553,177.981,14.635,151.506
C08041=1103.264,161.948,435.532,177.985,14.635,151.505
C08042=1103.270,162.197,435.510,177.988,14.634,151.504
C08043=1103.275,162.446,435.488,177.992,14.633,151.503
C08044=1103.281,162.695,435.467,177.995,14.632,151.502
C08045=1103.286,162.944,435.445,177.999,14.632,151.501
C08046=1103.292,163.193,435.423,178.003,14.631,151.500
C08047=1103.298,163.443,435.401,178.006,14.630,151.499
C08048=1103.303,163.691,435.380,178.010,14.630,151.498
C08049=1103.309,163.941,435.357,178.014,14.629,151.497
C08050=1103.314,164.189,435.336,178.018,14.629,151.496
C08051=1103.319,164.439,435.314,178.021,14.627,151.495
C08052=1103.325,164.687,435.293,178.025,14.627,151.494
C08053=1103.330,164.937,435.270,178.028,14.626,151.493
C08054=1103.336,165.185,435.249,178.032,14.625,151.492
C08055=1103.341,165.435,435.227,178.036,14.625,151.491
C08056=1103.347,165.683,435.205,178.040,14.624,151.490
C08057=1103.353,165.932,435.183,178.043,14.623,151.489
C08058=1103.359,166.182,435.161,178.047,14.622,151.488
C08059=1103.364,166.430,435.139,178.051,14.622,151.487
C08060=1103.370,166.680,435.117,178.055,14.621,151.486
C08061=1103.375,166.928,435.096,178.059,14.621,151.485
C08062=1103.381,167.177,435.073,178.062,14.619,151.484
C08063=1103.387,167.426,435.051,178.066,14.619,151.483
C08064=1103.392,167.675,435.030,178.069,14.618,151.482
C08065=1103.398,167.925,435.008,178.073,14.617,151.481
C08066=1103.403,168.173,434.985,178.077,14.616,151.480
C08067=1103.409,168.422,434.963,178.081,14.616,151.479
C08068=1103.414,168.671,434.941,178.084,14.615,151.478
C08069=1103.421,168.920,434.919,178.088,14.614,151.477
C08070=1103.426,169.169,434.897,178.091,14.613,151.476
C08071=1103.432,169.418,434.875,178.096,14.612,151.475
C08072=1103.437,169.668,434.853,178.100,14.612,151.474
C08073=1103.442,169.916,434.830,178.103,14.611,151.473
C08074=1103.449,170.165,434.809,178.107,14.610,151.472
C08075=1103.454,170.414,434.786,178.110,14.609,151.471
C08076=1103.459,170.663,434.764,178.115,14.608,151.470
C08077=1103.465,170.912,434.742,178.118,14.607,151.469
C08078=1103.471,171.161,434.719,178.122,14.607,151.468
C08079=1103.477,171.409,434.698,178.126,14.606,151.467
C08080=1103.482,171.658,434.675,178.130,14.605,151.466
C08081=1103.488,171.908,434.653,178.133,14.604,151.465
C08082=1103.494,172.157,434.631,178.137,14.603,151.464
C08083=1103.499,172.405,434.609,178.141,14.602,151.463
C08084=1103.504,172.655,434.587,178.145,14.602,151.462
C08085=1103.511,172.903,434.564,178.149,14.601,151.461
C08086=1103.516,173.153,434.542,178.152,14.600,151.460
C08087=1103.521,173.401,434.519,178.156,14.599,151.459
C08088=1103.528,173.650,434.498,178.160,14.598,151.458
C08089=1103.533,173.899,434.475,178.164,14.598,151.457
C08090=1103.539,174.149,434.453,178.167,14.596,151.456
C08091=1103.545,174.396,434.431,178.172,14.596,151.455
C08092=1103.550,174.646,434.408,178.175,14.594,151.454
C08093=1103.556,174.895,434.385,178.179,14.594,151.453
C08094=1103.561,175.144,434.362,178.182,14.593,151.452
C08095=1103.568,175.393,434.341,178.187,14.592,151.451
C08096=1103.573,175.641,434.318,178.190,14.591,151.450
C08097=1103.579,175.913,434.293,178.194,14.590,151.449
C08098=1103.585,176.185,434.269,178.199,14.589,151.447
C08099=1103.592,176.457,434.245,178.203,14.589,151.446
C08100=1103.598,176.729,434.221,178.207,14.588,151.445
C08101=1103.604,176.978,434.198,178.211,14.587,151.444
C08102=1103.609,177.227,434.175,178.215,14.586,151.443
C08103=1103.615,177.476,434.152,178.219,14.585,151.442
C08104=1103.621,177.725,434.130,178.223,14.584,151.441
C08105=1103.627,177.974,434.107,178.226,14.583,151.440
C08106=1103.632,178.223,434.085,178.230,14.582,151.439
C08107=1103.637,178.471,434.062,178.234,14.581,151.438
C08108=1103.643,178.720,434.039,178.238,14.580,151.437
C08109=1103.650,178.969,434.017,178.242,14.579,151.436
C08110=1103.655,179.218,433.995,178.246,14.578,151.434
C08111=1103.661,179.467,433.972,178.249,14.577,151.433
C08112=1103.667,179.716,433.949,178.254,14.576,151.432
C08113=1103.672,179.965,433.926,178.258,14.576,151.431
C08114=1103.679,180.214,433.904,178.261,14.574,151.430
C08115=1103.684,180.463,433.881,178.266,14.574,151.429
C08116=1103.690,180.712,433.858,178.269,14.572,151.428
C08117=1103.696,180.961,433.836,178.273,14.572,151.427
C08118=1103.701,181.210,433.813,178.277,14.570,151.426
C08119=1103.707,181.459,433.790,178.281,14.570,151.425
C08120=1103.713,181.707,433.768,178.284,14.568,151.424
C08121=1103.719,181.956,433.745,178.289,14.568,151.423
C08122=1103.724,182.204,433.722,178.292,14.567,151.422
C08123=1103.730,182.453,433.699,178.296,14.566,151.421
C08124=1103.736,182.703,433.677,178.300,14.565,151.420
C08125=1103.741,182.952,433.654,178.304,14.564,151.418
C08126=1103.747,183.201,433.631,178.309,14.563,151.417
C08127=1103.753,183.450,433.608,178.312,14.562,151.416
C08128=1103.759,183.698,433.585,178.316,14.561,151.415
C08129=1103.765,183.947,433.562,178.320,14.560,151.414
C08130=1103.771,184.196,433.540,178.324,14.559,151.413
C08131=1103.776,184.445,433.517,178.327,14.558,151.412
C08132=1103.782,184.694,433.494,178.332,14.557,151.411
C08133=1103.788,184.943,433.470,178.336,14.555,151.410
C08134=1103.794,185.192,433.447,178.340,14.555,151.409
C08135=1103.800,185.440,433.424,178.343,14.553,151.407
C08136=1103.805,185.689,433.401,178.347,14.553,151.406
C08137=1103.810,185.938,433.378,178.352,14.552,151.405
C08138=1103.816,186.187,433.355,178.355,14.551,151.404
C08139=1103.822,186.436,433.332,178.359,14.550,151.403
C08140=1103.828,186.685,433.309,178.363,14.549,151.402
C08141=1103.833,186.933,433.286,178.367,14.548,151.401
C08142=1103.838,187.183,433.262,178.371,14.547,151.400
C08143=1103.844,187.432,433.239,178.375,14.547,151.399
C08144=1103.850,187.680,433.216,178.379,14.545,151.398
C08145=1103.855,187.929,433.193,178.383,14.544,151.397
C08146=1103.862,188.178,433.170,178.387,14.544,151.396
C08147=1103.867,188.427,433.146,178.391,14.542,151.395
C08148=1103.872,188.676,433.123,178.395,14.542,151.393
C08149=1103.878,188.925,433.100,178.398,14.540,151.392
C08150=1103.884,189.174,433.077,178.402,14.540,151.391
C08151=1103.889,189.422,433.053,178.406,14.538,151.390
C08152=1103.895,189.671,433.030,178.410,14.537,151.389
C08153=1103.900,189.920,433.007,178.415,14.537,151.388
C08154=1103.906,190.169,432.984,178.418,14.536,151.387
C08155=1103.912,190.417,432.960,178.422,14.535,151.386
C08156=1103.917,190.666,432.937,178.426,14.534,151.385
C08157=1103.923,190.915,432.914,178.430,14.533,151.384
C08158=1103.928,191.164,432.891,178.434,14.531,151.382
C08159=1103.934,191.413,432.867,178.438,14.531,151.381
C08160=1103.940,191.662,432.844,178.442,14.530,151.380
C08161=1103.946,191.934,432.818,178.446,14.528,151.379
C08162=1103.952,192.205,432.792,178.451,14.527,151.378
C08163=1103.959,192.476,432.767,178.455,14.526,151.377
C08164=1103.964,192.748,432.741,178.460,14.525,151.375
C08165=1103.970,192.997,432.718,178.463,14.524,151.374
C08166=1103.976,193.246,432.695,178.468,14.524,151.373
C08167=1103.981,193.494,432.671,178.471,14.522,151.372
C08168=1103.987,193.743,432.648,178.476,14.521,151.371
C08169=1103.993,193.992,432.625,178.480,14.521,151.370
C08170=1103.998,194.241,432.600,178.484,14.519,151.369
C08171=1104.005,194.490,432.577,178.488,14.518,151.368
C08172=1104.011,194.738,432.553,178.491,14.517,151.367
C08173=1104.016,194.988,432.530,178.496,14.516,151.365
C08174=1104.022,195.236,432.506,178.499,14.515,151.364
C08175=1104.027,195.485,432.483,178.504,14.514,151.363
C08176=1104.033,195.733,432.459,178.507,14.512,151.362
C08177=1104.039,195.983,432.436,178.512,14.512,151.361
C08178=1104.044,196.232,432.411,178.516,14.511,151.360
C08179=1104.050,196.481,432.388,178.520,14.510,151.359
C08180=1104.055,196.729,432.364,178.524,14.509,151.358
C08181=1104.061,196.977,432.341,178.528,14.507,151.356
C08182=1104.068,197.227,432.317,178.532,14.507,151.355
C08183=1104.073,197.476,432.293,178.536,14.505,151.354
C08184=1104.079,197.724,432.270,178.540,14.504,151.353
C08185=1104.084,197.973,432.246,178.545,14.503,151.352
C08186=1104.090,198.221,432.222,178.548,14.502,151.351
C08187=1104.096,198.471,432.198,178.553,14.501,151.349
C08188=1104.102,198.719,432.175,178.556,14.500,151.348
C08189=1104.107,198.968,432.150,178.561,14.499,151.347
C08190=1104.113,199.217,432.127,178.564,14.498,151.346
C08191=1104.119,199.466,432.103,178.569,14.497,151.345
C08192=1104.125,199.715,432.079,178.572,14.495,151.344
C08193=1104.130,199.964,432.056,178.577,14.494,151.343
C08194=1104.136,200.213,432.032,178.581,14.494,151.341
C08195=1104.142,200.461,432.007,178.585,14.492,151.340
C08196=1104.148,200.710,431.984,178.589,14.492,151.339
C08197=1104.153,200.958,431.959,178.593,14.490,151.338
C08198=1104.159,201.208,431.936,178.597,14.489,151.337
C08199=1104.165,201.456,431.912,178.601,14.488,151.336
C08200=1104.171,201.705,431.888,178.605,14.487,151.334
C08201=1104.176,201.954,431.863,178.610,14.486,151.333
C08202=1104.183,202.202,431.840,178.613,14.484,151.332
C08203=1104.187,202.451,431.816,178.618,14.484,151.331
C08204=1104.194,202.700,431.792,178.621,14.482,151.330
C08205=1104.199,202.949,431.768,178.626,14.481,151.329
C08206=1104.205,203.198,431.744,178.629,14.480,151.328
C08207=1104.211,203.447,431.720,178.634,14.479,151.326
C08208=1104.217,203.695,431.695,178.638,14.478,151.325
C08209=1104.222,203.944,431.671,178.642,14.477,151.324
C08210=1104.228,204.192,431.648,178.646,14.476,151.323
C08211=1104.234,204.442,431.624,178.650,14.474,151.322
C08212=1104.239,204.691,431.599,178.654,14.474,151.321
C08213=1104.244,204.939,431.575,178.658,14.472,151.319
C08214=1104.251,205.188,431.551,178.663,14.471,151.318
C08215=1104.256,205.437,431.527,178.667,14.471,151.317
C08216=1104.261,205.685,431.503,178.671,14.469,151.316
C08217=1104.267,205.935,431.478,178.675,14.468,151.315
C08218=1104.273,206.183,431.454,178.679,14.467,151.314
C08219=1104.279,206.432,431.430,178.683,14.466,151.312
C08220=1104.285,206.681,431.405,178.687,14.465,151.311
C08221=1104.290,206.929,431.381,178.691,14.464,151.310
C08222=1104.297,207.178,431.357,178.696,14.463,151.309
C08223=1104.302,207.426,431.332,178.699,14.461,151.308
C08224=1104.307,207.675,431.308,178.704,14.460,151.307
C08225=1104.330,208.673,431.211,178.732,14.462,151.301
C08226=1104.338,209.041,431.174,178.737,14.461,151.299
C08227=1104.347,209.407,431.138,178.743,14.462,151.298
C08228=1104.356,209.774,431.102,178.749,14.461,151.297
C08229=1104.364,210.142,431.065,178.755,14.460,151.295
C08230=1104.370,210.390,431.041,178.758,14.460,151.294
C08231=1104.376,210.640,431.017,178.762,14.460,151.293
C08232=1104.381,210.888,430.992,178.766,14.460,151.293
C08233=1104.387,211.136,430.967,178.770,14.459,151.292
C08234=1104.392,211.386,430.943,178.774,14.458,151.291
C08235=1104.398,211.634,430.918,178.777,14.458,151.290
C08236=1104.404,211.883,430.893,178.781,14.458,151.289
C08237=1104.409,212.131,430.869,178.785,14.458,151.288
C08238=1104.415,212.381,430.844,178.789,14.458,151.287
C08239=1104.421,212.629,430.819,178.793,14.457,151.286
C08240=1104.427,212.878,430.795,178.797,14.457,151.285
C08241=1104.432,213.126,430.769,178.800,14.457,151.284
C08242=1104.437,213.376,430.744,178.804,14.456,151.283
C08243=1104.443,213.624,430.720,178.808,14.456,151.282
C08244=1104.449,213.873,430.695,178.812,14.456,151.281
C08245=1104.454,214.121,430.671,178.816,14.456,151.280
C08246=1104.460,214.370,430.645,178.820,14.456,151.280
C08247=1104.466,214.619,430.621,178.824,14.455,151.279
C08248=1104.472,214.868,430.596,178.828,14.455,151.278
C08249=1104.477,215.116,430.571,178.832,14.455,151.277
C08250=1104.482,215.365,430.546,178.835,14.454,151.276
C08251=1104.488,215.613,430.521,178.839,14.454,151.275
C08252=1104.494,215.863,430.497,178.843,14.454,151.274
C08253=1104.500,216.111,430.472,178.847,14.454,151.273
C08254=1104.505,216.360,430.447,178.851,14.454,151.272
C08255=1104.511,216.609,430.421,178.855,14.453,151.271
C08256=1104.516,216.857,430.396,178.859,14.453,151.271
C08257=1104.522,217.106,430.371,178.863,14.453,151.269
C08258=1104.528,217.354,430.347,178.867,14.453,151.269
C08259=1104.533,217.604,430.321,178.870,14.452,151.268
C08260=1104.539,217.852,430.296,178.874,14.452,151.267
C08261=1104.545,218.100,430.271,178.878,14.452,151.266
C08262=1104.551,218.350,430.246,178.882,14.452,151.265
C08263=1104.556,218.598,430.221,178.886,14.451,151.264
C08264=1104.562,218.847,430.195,178.890,14.451,151.263
C08265=1104.567,219.095,430.171,178.894,14.451,151.262
C08266=1104.573,219.344,430.146,178.897,14.451,151.261
C08267=1104.579,219.593,430.120,178.901,14.451,151.260
C08268=1104.584,219.841,430.096,178.905,14.450,151.260
C08269=1104.590,220.090,430.070,178.909,14.450,151.258
C08270=1104.597,220.339,430.045,178.913,14.449,151.258
C08271=1104.601,220.588,430.020,178.916,14.449,151.257
C08272=1104.607,220.836,429.995,178.920,14.449,151.256
C08273=1104.614,221.085,429.969,178.924,14.449,151.255
C08274=1104.618,221.333,429.944,178.928,14.449,151.254
C08275=1104.625,221.582,429.919,178.932,14.448,151.253
C08276=1104.631,221.831,429.894,178.936,14.448,151.252
C08277=1104.635,222.080,429.868,178.940,14.448,151.251
C08278=1104.644,222.450,429.831,178.946,14.447,151.250
C08279=1104.653,222.821,429.793,178.952,14.448,151.249
C08280=1104.660,223.192,429.755,178.957,14.447,151.247
C08281=1104.670,223.562,429.717,178.963,14.447,151.246
C08282=1104.675,223.810,429.692,178.967,14.447,151.245
C08283=1104.680,224.059,429.666,178.970,14.447,151.244
C08284=1104.687,224.308,429.641,178.975,14.446,151.243
C08285=1104.692,224.557,429.615,178.979,14.446,151.242
C08286=1104.698,224.805,429.590,178.982,14.446,151.241
C08287=1104.703,225.054,429.564,178.986,14.446,151.240
C08288=1104.709,225.303,429.539,178.990,14.446,151.240
C08289=1104.714,225.551,429.513,178.994,14.446,151.239
C08290=1104.720,225.800,429.488,178.998,14.446,151.238
C08291=1104.726,226.048,429.462,179.002,14.445,151.237
C08292=1104.732,226.297,429.437,179.006,14.445,151.236
C08293=1104.737,226.545,429.411,179.010,14.445,151.235
C08294=1104.743,226.794,429.386,179.013,14.445,151.234
C08295=1104.749,227.043,429.360,179.018,14.445,151.233
C08296=1104.754,227.292,429.334,179.021,14.444,151.232
C08297=1104.760,227.540,429.309,179.025,14.444,151.231
C08298=1104.765,227.788,429.282,179.029,14.444,151.231
C08299=1104.772,228.037,429.257,179.032,14.444,151.230
C08300=1104.777,228.286,429.231,179.036,14.444,151.229
C08301=1104.783,228.535,429.206,179.040,14.443,151.228
C08302=1104.788,228.783,429.180,179.044,14.443,151.227
C08303=1104.794,229.032,429.154,179.048,14.443,151.226
C08304=1104.800,229.281,429.129,179.052,14.443,151.225
C08305=1104.806,229.529,429.102,179.056,14.443,151.224
C08306=1104.811,229.778,429.076,179.060,14.443,151.223
C08307=1104.817,230.027,429.051,179.064,14.443,151.222
C08308=1104.822,230.275,429.025,179.068,14.442,151.221
C08309=1104.829,230.523,428.999,179.072,14.442,151.221
C08310=1104.834,230.772,428.973,179.076,14.442,151.220
C08311=1104.840,231.021,428.948,179.079,14.442,151.219
C08312=1104.845,231.270,428.922,179.083,14.442,151.218
C08313=1104.852,231.518,428.896,179.087,14.442,151.217
C08314=1104.856,231.766,428.870,179.091,14.442,151.216
C08315=1104.862,232.015,428.844,179.095,14.442,151.215
C08316=1104.867,232.264,428.818,179.099,14.442,151.214
C08317=1104.874,232.512,428.792,179.103,14.442,151.214
C08318=1104.879,232.761,428.766,179.107,14.442,151.213
C08319=1104.885,233.010,428.740,179.110,14.442,151.212
C08320=1104.891,233.259,428.714,179.114,14.442,151.211
C08321=1104.895,233.507,428.688,179.118,14.442,151.210
C08322=1104.902,233.755,428.662,179.122,14.441,151.209
C08323=1104.907,234.004,428.636,179.126,14.441,151.208
C08324=1104.913,234.253,428.610,179.130,14.441,151.207
C08325=1104.919,234.501,428.583,179.134,14.441,151.206
C08326=1104.924,234.750,428.557,179.138,14.441,151.206
C08327=1104.930,234.999,428.531,179.141,14.441,151.205
C08328=1104.935,235.248,428.505,179.145,14.441,151.204
C08329=1104.942,235.496,428.479,179.149,14.441,151.203
C08330=1104.950,235.858,428.441,179.155,14.441,151.202
C08331=1104.958,236.220,428.403,179.161,14.441,151.200
C08332=1104.966,236.583,428.365,179.166,14.441,151.199
C08333=1104.974,236.944,428.327,179.171,14.440,151.198
C08334=1104.980,237.192,428.300,179.175,14.440,151.197
C08335=1104.985,237.441,428.274,179.179,14.440,151.196
C08336=1104.991,237.690,428.247,179.183,14.440,151.195
C08337=1104.997,237.939,428.221,179.187,14.440,151.194
C08338=1105.002,238.187,428.195,179.191,14.440,151.193
C08339=1105.008,238.435,428.168,179.195,14.440,151.193
C08340=1105.014,238.684,428.142,179.199,14.441,151.192
C08341=1105.019,238.933,428.116,179.203,14.440,151.191
C08342=1105.025,239.181,428.089,179.207,14.440,151.190
C08343=1105.031,239.430,428.063,179.211,14.440,151.189
C08344=1105.036,239.678,428.036,179.215,14.440,151.188
C08345=1105.042,239.927,428.010,179.219,14.440,151.187
C08346=1105.048,240.176,427.984,179.223,14.440,151.186
C08347=1105.053,240.424,427.957,179.227,14.440,151.186
C08348=1105.059,240.672,427.931,179.230,14.440,151.185
C08349=1105.065,240.921,427.904,179.234,14.440,151.184
C08350=1105.070,241.170,427.878,179.238,14.440,151.183
C08351=1105.076,241.418,427.851,179.242,14.440,151.182
C08352=1105.082,241.666,427.825,179.246,14.440,151.181
C08353=1105.088,241.915,427.798,179.249,14.440,151.180
C08354=1105.093,242.164,427.770,179.253,14.440,151.180
C08355=1105.099,242.413,427.744,179.257,14.440,151.179
C08356=1105.105,242.662,427.718,179.261,14.440,151.178
C08357=1105.110,242.910,427.691,179.265,14.440,151.177
C08358=1105.116,243.158,427.664,179.269,14.440,151.176
C08359=1105.122,243.407,427.638,179.273,14.440,151.175
C08360=1105.128,243.655,427.611,179.277,14.440,151.174
C08361=1105.134,243.903,427.585,179.280,14.440,151.173
C08362=1105.139,244.152,427.557,179.284,14.440,151.173
C08363=1105.144,244.400,427.531,179.288,14.440,151.172
C08364=1105.150,244.649,427.504,179.292,14.441,151.171
C08365=1105.156,244.898,427.478,179.296,14.441,151.170
C08366=1105.161,245.146,427.451,179.300,14.441,151.169
C08367=1105.167,245.395,427.424,179.304,14.441,151.168
C08368=1105.173,245.644,427.397,179.308,14.441,151.167
C08369=1105.179,245.892,427.371,179.312,14.441,151.167
C08370=1105.184,246.141,427.343,179.315,14.441,151.166
C08371=1105.189,246.389,427.317,179.319,14.441,151.165
C08372=1105.195,246.637,427.289,179.323,14.441,151.164
C08373=1105.201,246.885,427.263,179.327,14.441,151.163
C08374=1105.206,247.134,427.235,179.331,14.441,151.162
C08375=1105.212,247.382,427.209,179.335,14.441,151.162
C08376=1105.218,247.631,427.182,179.338,14.441,151.161
C08377=1105.223,247.880,427.154,179.342,14.441,151.160
C08378=1105.229,248.128,427.128,179.347,14.442,151.159
C08379=1105.234,248.377,427.101,179.351,14.442,151.158
C08380=1105.240,248.625,427.074,179.354,14.442,151.157
C08381=1105.245,248.874,427.047,179.358,14.442,151.157
C08382=1105.254,249.229,427.008,179.363,14.442,151.155
C08383=1105.262,249.584,426.969,179.369,14.442,151.154
C08384=1105.269,249.940,426.930,179.375,14.442,151.153
C08385=1105.278,250.296,426.892,179.380,14.443,151.152
C08386=1105.283,250.544,426.864,179.384,14.443,151.151
C08387=1105.289,250.792,426.837,179.388,14.443,151.150
C08388=1105.295,251.041,426.810,179.392,14.443,151.149
C08389=1105.300,251.290,426.783,179.395,14.443,151.149
C08390=1105.306,251.538,426.756,179.399,14.443,151.148
C08391=1105.311,251.786,426.728,179.403,14.443,151.147
C08392=1105.317,252.034,426.702,179.407,14.443,151.146
C08393=1105.323,252.284,426.674,179.411,14.444,151.145
C08394=1105.329,252.532,426.647,179.415,14.444,151.144
C08395=1105.334,252.780,426.619,179.419,14.444,151.144
C08396=1105.339,253.029,426.592,179.423,14.445,151.143
C08397=1105.345,253.277,426.564,179.427,14.445,151.142
C08398=1105.350,253.526,426.537,179.430,14.444,151.141
C08399=1105.357,253.774,426.510,179.434,14.444,151.140
C08400=1105.362,254.022,426.482,179.438,14.445,151.139
C08401=1105.368,254.271,426.455,179.442,14.445,151.139
C08402=1105.373,254.520,426.428,179.446,14.445,151.138
C08403=1105.379,254.768,426.401,179.450,14.445,151.137
C08404=1105.384,255.016,426.373,179.454,14.446,151.136
C08405=1105.390,255.265,426.345,179.458,14.446,151.135
C08406=1105.396,255.513,426.318,179.461,14.446,151.134
C08407=1105.401,255.762,426.291,179.465,14.446,151.134
C08408=1105.408,256.010,426.263,179.469,14.446,151.133
C08409=1105.413,256.258,426.235,179.473,14.446,151.132
C08410=1105.418,256.507,426.208,179.477,14.447,151.131
C08411=1105.425,256.755,426.180,179.481,14.447,151.130
C08412=1105.430,257.004,426.153,179.485,14.447,151.130
C08413=1105.436,257.252,426.125,179.489,14.447,151.129
C08414=1105.442,257.501,426.098,179.492,14.448,151.128
C08415=1105.447,257.749,426.070,179.496,14.448,151.127
C08416=1105.453,257.997,426.043,179.500,14.448,151.126
C08417=1105.459,258.246,426.015,179.504,14.449,151.126
C08418=1105.464,258.494,425.987,179.508,14.449,151.125
C08419=1105.470,258.742,425.960,179.512,14.449,151.124
C08420=1105.476,258.991,425.932,179.516,14.449,151.123
C08421=1105.481,259.240,425.904,179.519,14.449,151.122
C08422=1105.488,259.488,425.876,179.523,14.449,151.121
C08423=1105.493,259.736,425.848,179.527,14.449,151.121
C08424=1105.498,259.985,425.821,179.531,14.450,151.120
C08425=1105.504,260.233,425.793,179.535,14.450,151.119
C08426=1105.510,260.481,425.765,179.539,14.450,151.118
C08427=1105.516,260.730,425.737,179.543,14.450,151.117
C08428=1105.522,260.978,425.709,179.546,14.450,151.117
C08429=1105.527,261.226,425.682,179.550,14.450,151.116
C08430=1105.533,261.475,425.654,179.555,14.451,151.115
C08431=1105.539,261.723,425.626,179.558,14.451,151.114
C08432=1105.545,261.972,425.598,179.562,14.451,151.113
C08433=1105.551,262.220,425.570,179.566,14.452,151.113
C08434=1105.559,262.573,425.531,179.572,14.452,151.111
C08435=1105.567,262.925,425.491,179.577,14.452,151.110
C08436=1105.575,263.278,425.451,179.582,14.452,151.109
C08437=1105.583,263.631,425.412,179.588,14.453,151.108
C08438=1105.589,263.880,425.383,179.592,14.453,151.107
C08439=1105.594,264.128,425.356,179.595,14.453,151.106
C08440=1105.601,264.376,425.328,179.600,14.454,151.105
C08441=1105.606,264.624,425.300,179.604,14.454,151.105
C08442=1105.612,264.873,425.272,179.607,14.454,151.104
C08443=1105.618,265.121,425.244,179.611,14.455,151.103
C08444=1105.624,265.370,425.215,179.615,14.455,151.102
C08445=1105.629,265.618,425.187,179.618,14.455,151.102
C08446=1105.635,265.866,425.159,179.623,14.456,151.101
C08447=1105.640,266.114,425.131,179.627,14.456,151.100
C08448=1105.646,266.363,425.103,179.630,14.456,151.099
C08449=1105.651,266.611,425.075,179.634,14.457,151.099
C08450=1105.658,266.859,425.046,179.638,14.457,151.098
C08451=1105.663,267.107,425.018,179.642,14.458,151.097
C08452=1105.669,267.356,424.989,179.646,14.458,151.096
C08453=1105.674,267.604,424.961,179.649,14.458,151.095
C08454=1105.680,267.853,424.933,179.653,14.458,151.095
C08455=1105.686,268.101,424.905,179.658,14.459,151.094
C08456=1105.692,268.350,424.877,179.661,14.459,151.093
C08457=1105.697,268.597,424.848,179.665,14.460,151.092
C08458=1105.702,268.846,424.819,179.669,14.460,151.091
C08459=1105.708,269.094,424.791,179.672,14.460,151.091
C08460=1105.714,269.343,424.763,179.677,14.461,151.090
C08461=1105.719,269.591,424.734,179.680,14.461,151.089
C08462=1105.725,269.839,424.706,179.684,14.462,151.088
C08463=1105.731,270.088,424.678,179.688,14.462,151.088
C08464=1105.737,270.336,424.650,179.691,14.462,151.087
C08465=1105.743,270.584,424.621,179.696,14.463,151.086
C08466=1105.748,270.832,424.593,179.700,14.463,151.085
C08467=1105.753,271.081,424.564,179.703,14.464,151.085
C08468=1105.759,271.329,424.535,179.707,14.464,151.084
C08469=1105.765,271.578,424.507,179.711,14.465,151.083
C08470=1105.771,271.826,424.478,179.715,14.465,151.082
C08471=1105.777,272.074,424.450,179.719,14.465,151.082
C08472=1105.782,272.323,424.421,179.722,14.466,151.081
C08473=1105.787,272.570,424.392,179.727,14.466,151.080
C08474=1105.793,272.819,424.364,179.730,14.467,151.079
C08475=1105.799,273.068,424.335,179.734,14.467,151.079
C08476=1105.805,273.315,424.307,179.738,14.467,151.078
C08477=1105.810,273.564,424.278,179.742,14.468,151.077
C08478=1105.816,273.812,424.249,179.745,14.469,151.076
C08479=1105.822,274.060,424.221,179.749,14.469,151.076
C08480=1105.828,274.309,424.192,179.753,14.469,151.075
C08481=1105.833,274.557,424.163,179.757,14.470,151.074
C08482=1105.839,274.805,424.134,179.761,14.470,151.073
C08483=1105.845,275.054,424.106,179.764,14.471,151.073
C08484=1105.850,275.301,424.077,179.768,14.471,151.072
C08485=1105.856,275.550,424.048,179.773,14.472,151.071
C08486=1105.864,275.906,424.007,179.777,14.472,151.070
C08487=1105.872,276.261,423.966,179.783,14.473,151.069
C08488=1105.880,276.617,423.924,179.789,14.474,151.068
C08489=1105.888,276.972,423.883,179.794,14.474,151.067
C08490=1105.894,277.220,423.854,179.798,14.476,151.066
C08491=1105.900,277.469,423.825,179.802,14.476,151.066
C08492=1105.905,277.717,423.796,179.805,14.476,151.065
C08493=1105.911,277.965,423.767,179.809,14.476,151.064
C08494=1105.917,278.213,423.738,179.813,14.478,151.063
C08495=1105.923,278.462,423.708,179.817,14.478,151.063
C08496=1105.928,278.710,423.680,179.820,14.478,151.062
C08497=1105.933,278.958,423.651,179.825,14.479,151.061
C08498=1105.940,279.206,423.622,179.828,14.480,151.060
C08499=1105.945,279.454,423.592,179.832,14.480,151.060
C08500=1105.951,279.703,423.564,179.835,14.480,151.059
C08501=1105.956,279.951,423.534,179.840,14.482,151.058
C08502=1105.962,280.199,423.505,179.843,14.482,151.058
C08503=1105.967,280.447,423.476,179.847,14.482,151.057
C08504=1105.973,280.695,423.447,179.851,14.483,151.056
C08505=1105.979,280.944,423.417,179.855,14.484,151.056
C08506=1105.985,281.192,423.389,179.858,14.484,151.055
C08507=1105.990,281.441,423.360,179.863,14.485,151.054
C08508=1105.996,281.688,423.331,179.866,14.486,151.053
C08509=1106.002,281.937,423.301,179.870,14.486,151.053
C08510=1106.008,282.185,423.272,179.873,14.486,151.052
C08511=1106.013,282.433,423.243,179.878,14.487,151.051
C08512=1106.018,282.681,423.213,179.881,14.488,151.051
C08513=1106.025,282.929,423.184,179.885,14.488,151.050
C08514=1106.030,283.178,423.155,179.889,14.489,151.049
C08515=1106.036,283.426,423.125,179.893,14.490,151.049
C08516=1106.041,283.673,423.096,179.896,14.490,151.048
C08517=1106.047,283.922,423.067,179.900,14.491,151.047
C08518=1106.052,284.170,423.037,179.904,14.492,151.046
C08519=1106.058,284.418,423.008,179.907,14.492,151.046
C08520=1106.064,284.667,422.978,179.912,14.493,151.045
C08521=1106.069,284.915,422.949,179.915,14.494,151.044
C08522=1106.075,285.163,422.920,179.919,14.494,151.044
C08523=1106.081,285.411,422.890,179.923,14.495,151.043
C08524=1106.086,285.660,422.861,179.926,14.496,151.042
C08525=1106.092,285.908,422.832,179.930,14.496,151.042
C08526=1106.098,286.156,422.801,179.934,14.497,151.041
C08527=1106.104,286.404,422.772,179.938,14.498,151.040
C08528=1106.109,286.653,422.742,179.941,14.498,151.040
C08529=1106.115,286.900,422.713,179.946,14.499,151.039
C08530=1106.120,287.148,422.684,179.949,14.500,151.038
C08531=1106.126,287.396,422.653,179.953,14.501,151.038
C08532=1106.132,287.645,422.624,179.957,14.501,151.037
C08533=1106.138,287.893,422.595,179.960,14.502,151.036
C08534=1106.143,288.141,422.565,179.965,14.503,151.036
C08535=1106.149,288.389,422.535,179.968,14.503,151.035
C08536=1106.155,288.638,422.505,179.972,14.504,151.034
C08537=1106.161,288.886,422.476,179.976,14.505,151.034
C08538=1106.169,289.250,422.433,179.981,14.506,151.033
C08539=1106.178,289.615,422.389,179.987,14.507,151.032
C08540=1106.186,289.980,422.345,179.992,14.508,151.031
C08541=1106.194,290.345,422.300,179.997,14.509,151.030
C08542=1106.200,290.594,422.271,-179.999,14.510,151.029
C08543=1106.206,290.842,422.242,-179.995,14.511,151.028
C08544=1106.212,291.090,422.211,-179.991,14.512,151.028
C08545=1106.217,291.338,422.182,-179.987,14.512,151.027
C08546=1106.223,291.586,422.151,-179.984,14.513,151.026
C08547=1106.228,291.834,422.122,-179.980,14.514,151.026
C08548=1106.234,292.082,422.091,-179.976,14.515,151.025
C08549=1106.240,292.331,422.062,-179.972,14.516,151.025
C08550=1106.245,292.578,422.032,-179.969,14.516,151.024
C08551=1106.250,292.826,422.002,-179.965,14.517,151.023
C08552=1106.256,293.074,421.972,-179.961,14.518,151.023
C08553=1106.262,293.322,421.942,-179.958,14.519,151.022
C08554=1106.268,293.570,421.912,-179.953,14.520,151.021
C08555=1106.273,293.819,421.882,-179.950,14.520,151.021
C08556=1106.279,294.066,421.852,-179.947,14.521,151.020
C08557=1106.284,294.315,421.822,-179.943,14.522,151.019
C08558=1106.290,294.563,421.792,-179.939,14.523,151.019
C08559=1106.296,294.811,421.761,-179.935,14.524,151.018
C08560=1106.302,295.059,421.732,-179.932,14.525,151.018
C08561=1106.307,295.307,421.701,-179.928,14.525,151.017
C08562=1106.313,295.555,421.672,-179.924,14.527,151.016
C08563=1106.319,295.804,421.641,-179.921,14.527,151.016
C08564=1106.325,296.052,421.611,-179.916,14.529,151.015
C08565=1106.331,296.299,421.580,-179.913,14.529,151.014
C08566=1106.337,296.548,421.551,-179.909,14.531,151.014
C08567=1106.342,296.796,421.520,-179.905,14.531,151.013
C08568=1106.347,297.044,421.490,-179.902,14.531,151.013
C08569=1106.353,297.292,421.460,-179.898,14.533,151.012
C08570=1106.359,297.540,421.430,-179.895,14.533,151.011
C08571=1106.365,297.788,421.399,-179.891,14.535,151.011
C08572=1106.370,298.036,421.369,-179.887,14.535,151.010
C08573=1106.376,298.284,421.338,-179.883,14.537,151.010
C08574=1106.381,298.532,421.308,-179.880,14.538,151.009
C08575=1106.387,298.780,421.278,-179.875,14.539,151.008
C08576=1106.393,299.028,421.248,-179.872,14.540,151.008
C08577=1106.398,299.276,421.217,-179.868,14.541,151.007
C08578=1106.404,299.524,421.186,-179.865,14.542,151.007
C08579=1106.409,299.772,421.156,-179.861,14.543,151.006
C08580=1106.414,300.020,421.125,-179.857,14.544,151.006
C08581=1106.420,300.268,421.095,-179.853,14.545,151.005
C08582=1106.426,300.516,421.065,-179.850,14.546,151.004
C08583=1106.431,300.765,421.034,-179.847,14.546,151.004
C08584=1106.437,301.013,421.003,-179.843,14.548,151.003
C08585=1106.443,301.261,420.973,-179.839,14.548,151.003
C08586=1106.448,301.509,420.942,-179.835,14.550,151.002
C08587=1106.454,301.757,420.912,-179.832,14.551,151.002
C08588=1106.460,302.004,420.881,-179.828,14.552,151.001
C08589=1106.465,302.252,420.850,-179.825,14.553,151.001
C08590=1106.474,302.631,420.803,-179.818,14.555,151.000
C08591=1106.482,303.010,420.757,-179.813,14.556,150.999
C08592=1106.491,303.389,420.710,-179.807,14.558,150.998
C08593=1106.500,303.768,420.663,-179.802,14.560,150.997
C08594=1106.505,304.016,420.632,-179.799,14.561,150.997
C08595=1106.511,304.264,420.601,-179.794,14.562,150.996
C08596=1106.516,304.512,420.570,-179.791,14.563,150.995
C08597=1106.522,304.760,420.540,-179.787,14.564,150.995
C08598=1106.528,305.008,420.508,-179.784,14.565,150.994
C08599=1106.533,305.256,420.478,-179.780,14.566,150.994
C08600=1106.538,305.504,420.447,-179.776,14.568,150.993
C08601=1106.545,305.752,420.416,-179.773,14.569,150.993
C08602=1106.551,306.000,420.386,-179.769,14.570,150.992
C08603=1106.556,306.248,420.354,-179.765,14.571,150.992
C08604=1106.562,306.495,420.324,-179.762,14.572,150.991
C08605=1106.568,306.744,420.293,-179.758,14.573,150.990
C08606=1106.573,306.992,420.262,-179.754,14.574,150.990
C08607=1106.579,307.240,420.231,-179.751,14.575,150.989
C08608=1106.585,307.487,420.200,-179.747,14.577,150.989
C08609=1106.590,307.736,420.169,-179.744,14.578,150.988
C08610=1106.596,307.984,420.137,-179.740,14.579,150.988
C08611=1106.601,308.232,420.107,-179.736,14.580,150.987
C08612=1106.607,308.480,420.076,-179.733,14.581,150.987
C08613=1106.613,308.728,420.045,-179.729,14.583,150.986
C08614=1106.618,308.976,420.014,-179.725,14.583,150.986
C08615=1106.624,309.223,419.983,-179.721,14.585,150.985
C08616=1106.630,309.472,419.951,-179.718,14.586,150.985
C08617=1106.636,309.720,419.921,-179.714,14.587,150.984
C08618=1106.641,309.967,419.889,-179.711,14.588,150.984
C08619=1106.647,310.216,419.858,-179.707,14.590,150.983
C08620=1106.653,310.463,419.827,-179.704,14.590,150.982
C08621=1106.658,310.711,419.796,-179.700,14.592,150.982
C08622=1106.665,310.959,419.765,-179.696,14.593,150.981
C08623=1106.670,311.207,419.734,-179.693,14.594,150.981
C08624=1106.675,311.455,419.702,-179.689,14.596,150.981
C08625=1106.682,311.703,419.671,-179.686,14.597,150.980
C08626=1106.687,311.951,419.640,-179.682,14.598,150.980
C08627=1106.693,312.199,419.608,-179.678,14.599,150.979
C08628=1106.699,312.447,419.577,-179.675,14.601,150.979
C08629=1106.704,312.694,419.546,-179.671,14.602,150.978
C08630=1106.710,312.943,419.514,-179.667,14.603,150.977
C08631=1106.716,313.190,419.483,-179.663,14.604,150.977
C08632=1106.722,313.439,419.451,-179.660,14.605,150.976
C08633=1106.727,313.687,419.420,-179.656,14.607,150.976
C08634=1106.733,313.934,419.389,-179.653,14.608,150.975
C08635=1106.739,314.182,419.357,-179.649,14.609,150.975
C08636=1106.744,314.430,419.326,-179.646,14.610,150.974
C08637=1106.751,314.678,419.295,-179.642,14.612,150.974
C08638=1106.757,314.926,419.263,-179.638,14.613,150.973
C08639=1106.762,315.175,419.232,-179.635,14.614,150.973
C08640=1106.768,315.422,419.200,-179.631,14.616,150.972
C08641=1106.774,315.670,419.168,-179.628,14.617,150.972
C08642=1106.782,316.051,419.120,-179.622,14.619,150.971
C08643=1106.791,316.433,419.071,-179.616,14.622,150.971
C08644=1106.799,316.814,419.023,-179.612,14.624,150.970
C08645=1106.808,317.196,418.974,-179.606,14.626,150.969
C08646=1106.813,317.444,418.942,-179.603,14.627,150.969
C08647=1106.819,317.691,418.910,-179.599,14.629,150.968
C08648=1106.825,317.940,418.878,-179.595,14.631,150.968
C08649=1106.830,318.187,418.847,-179.592,14.632,150.968
C08650=1106.836,318.436,418.815,-179.588,14.633,150.967
C08651=1106.841,318.683,418.784,-179.585,14.635,150.967
C08652=1106.847,318.932,418.752,-179.581,14.636,150.966
C08653=1106.853,319.179,418.720,-179.578,14.638,150.966
C08654=1106.859,319.427,418.688,-179.574,14.640,150.966
C08655=1106.864,319.675,418.656,-179.571,14.641,150.965
C08656=1106.870,319.923,418.624,-179.567,14.642,150.965
C08657=1106.875,320.171,418.593,-179.563,14.644,150.964
C08658=1106.881,320.419,418.560,-179.560,14.645,150.964
C08659=1106.886,320.667,418.528,-179.557,14.647,150.963
C08660=1106.892,320.915,418.496,-179.553,14.649,150.963
C08661=1106.897,321.162,418.465,-179.550,14.650,150.963
C08662=1106.903,321.411,418.433,-179.546,14.651,150.962
C08663=1106.909,321.658,418.401,-179.542,14.653,150.962
C08664=1106.915,321.906,418.369,-179.539,14.654,150.961
C08665=1106.920,322.154,418.337,-179.536,14.656,150.961
C08666=1106.926,322.402,418.305,-179.532,14.658,150.961
C08667=1106.932,322.650,418.272,-179.529,14.659,150.960
C08668=1106.937,322.897,418.240,-179.525,14.661,150.960
C08669=1106.943,323.146,418.208,-179.521,14.663,150.959
C08670=1106.948,323.393,418.177,-179.518,14.664,150.959
C08671=1106.954,323.641,418.145,-179.515,14.666,150.959
C08672=1106.960,323.889,418.113,-179.511,14.667,150.958
C08673=1106.965,324.137,418.080,-179.508,14.668,150.958
C08674=1106.971,324.385,418.048,-179.504,14.670,150.958
C08675=1106.977,324.633,418.016,-179.501,14.672,150.957
C08676=1106.983,324.881,417.984,-179.498,14.673,150.957
C08677=1106.989,325.129,417.952,-179.494,14.675,150.956
C08678=1106.994,325.376,417.919,-179.490,14.677,150.956
C08679=1107.000,325.624,417.887,-179.487,14.679,150.956
C08680=1107.006,325.873,417.855,-179.483,14.680,150.955
C08681=1107.011,326.119,417.823,-179.480,14.682,150.955
C08682=1107.017,326.368,417.790,-179.476,14.683,150.954
C08683=1107.022,326.616,417.758,-179.472,14.685,150.954
C08684=1107.028,326.863,417.725,-179.470,14.687,150.954
C08685=1107.034,327.111,417.693,-179.466,14.688,150.953
C08686=1107.039,327.360,417.661,-179.462,14.690,150.953
C08687=1107.045,327.607,417.628,-179.459,14.691,150.953
C08688=1107.051,327.855,417.596,-179.456,14.693,150.952
C08689=1107.057,328.103,417.563,-179.452,14.695,150.952
C08690=1107.063,328.351,417.531,-179.448,14.697,150.952
C08691=1107.068,328.598,417.499,-179.445,14.698,150.951
C08692=1107.074,328.846,417.467,-179.442,14.700,150.951
C08693=1107.080,329.094,417.433,-179.438,14.702,150.950
C08694=1107.088,329.469,417.385,-179.433,14.705,150.950
C08695=1107.097,329.843,417.336,-179.428,14.707,150.949
C08696=1107.106,330.218,417.286,-179.422,14.710,150.949
C08697=1107.115,330.592,417.237,-179.417,14.713,150.948
C08698=1107.120,330.839,417.205,-179.414,14.714,150.948
C08699=1107.126,331.088,417.172,-179.411,14.716,150.948
C08700=1107.132,331.335,417.139,-179.407,14.718,150.947
C08701=1107.138,331.583,417.107,-179.403,14.720,150.947
C08702=1107.143,331.831,417.074,-179.400,14.721,150.947
C08703=1107.150,332.079,417.041,-179.397,14.723,150.946
C08704=1107.155,332.326,417.008,-179.393,14.725,150.946
C08705=1107.161,332.574,416.976,-179.390,14.727,150.946
C08706=1107.166,332.822,416.943,-179.386,14.729,150.945
C08707=1107.172,333.070,416.910,-179.383,14.731,150.945
C08708=1107.177,333.318,416.878,-179.380,14.732,150.945
C08709=1107.183,333.565,416.845,-179.376,14.734,150.945
C08710=1107.189,333.813,416.812,-179.373,14.736,150.944
C08711=1107.194,334.062,416.779,-179.369,14.738,150.944
C08712=1107.201,334.309,416.747,-179.366,14.740,150.944
C08713=1107.205,334.556,416.714,-179.363,14.742,150.943
C08714=1107.212,334.804,416.681,-179.359,14.744,150.943
C08715=1107.217,335.052,416.648,-179.356,14.746,150.943
C08716=1107.223,335.300,416.615,-179.353,14.748,150.943
C08717=1107.229,335.548,416.582,-179.349,14.750,150.942
C08718=1107.234,335.796,416.549,-179.346,14.752,150.942
C08719=1107.239,336.043,416.516,-179.342,14.754,150.942
C08720=1107.246,336.291,416.483,-179.339,14.756,150.942
C08721=1107.251,336.539,416.450,-179.336,14.758,150.941
C08722=1107.257,336.787,416.416,-179.332,14.760,150.941
C08723=1107.263,337.034,416.384,-179.329,14.762,150.941
C08724=1107.269,337.282,416.350,-179.326,14.764,150.941
C08725=1107.274,337.531,416.318,-179.322,14.766,150.940
C08726=1107.280,337.778,416.285,-179.318,14.768,150.940
C08727=1107.285,338.025,416.252,-179.315,14.770,150.940
C08728=1107.291,338.273,416.219,-179.312,14.772,150.940
C08729=1107.296,338.521,416.185,-179.309,14.774,150.939
C08730=1107.303,338.769,416.153,-179.306,14.776,150.939
C08731=1107.308,339.017,416.119,-179.302,14.778,150.939
C08732=1107.314,339.264,416.085,-179.299,14.780,150.939
C08733=1107.319,339.512,416.052,-179.295,14.782,150.938
C08734=1107.325,339.760,416.019,-179.292,14.785,150.938
C08735=1107.331,340.007,415.986,-179.288,14.787,150.938
C08736=1107.337,340.255,415.952,-179.285,14.789,150.938
C08737=1107.342,340.502,415.919,-179.282,14.791,150.938
C08738=1107.347,340.750,415.886,-179.279,14.793,150.937
C08739=1107.353,340.998,415.853,-179.276,14.795,150.937
C08740=1107.358,341.246,415.819,-179.272,14.797,150.937
C08741=1107.364,341.493,415.785,-179.269,14.799,150.937
C08742=1107.371,341.741,415.753,-179.266,14.802,150.937
C08743=1107.376,341.989,415.719,-179.262,14.804,150.936
C08744=1107.382,342.237,415.686,-179.259,14.806,150.936
C08745=1107.387,342.485,415.653,-179.256,14.808,150.936
C08746=1107.396,342.852,415.602,-179.251,14.812,150.936
C08747=1107.405,343.221,415.553,-179.246,14.815,150.935
C08748=1107.413,343.589,415.503,-179.241,14.819,150.935
C08749=1107.421,343.958,415.453,-179.236,14.822,150.935
C08750=1107.427,344.206,415.419,-179.232,14.824,150.935
C08751=1107.433,344.453,415.385,-179.230,14.826,150.935
C08752=1107.438,344.701,415.352,-179.226,14.828,150.934
C08753=1107.444,344.948,415.318,-179.223,14.830,150.934
C08754=1107.450,345.196,415.285,-179.220,14.833,150.934
C08755=1107.455,345.444,415.251,-179.217,14.835,150.934
C08756=1107.461,345.691,415.217,-179.213,14.838,150.934
C08757=1107.466,345.939,415.184,-179.210,14.840,150.934
C08758=1107.472,346.187,415.150,-179.207,14.842,150.934
C08759=1107.478,346.434,415.117,-179.204,14.845,150.933
C08760=1107.484,346.682,415.083,-179.200,14.847,150.933
C08761=1107.489,346.930,415.049,-179.197,14.849,150.933
C08762=1107.495,347.177,415.015,-179.194,14.852,150.933
C08763=1107.501,347.425,414.982,-179.191,14.854,150.933
C08764=1107.507,347.672,414.948,-179.187,14.857,150.933
C08765=1107.511,347.920,414.914,-179.184,14.860,150.933
C08766=1107.517,348.168,414.880,-179.180,14.862,150.933
C08767=1107.523,348.415,414.846,-179.177,14.864,150.932
C08768=1107.529,348.663,414.812,-179.174,14.867,150.932
C08769=1107.535,348.911,414.779,-179.171,14.869,150.932
C08770=1107.541,349.159,414.745,-179.168,14.872,150.932
C08771=1107.546,349.406,414.710,-179.164,14.874,150.932
C08772=1107.551,349.654,414.677,-179.161,14.877,150.932
C08773=1107.557,349.901,414.643,-179.158,14.879,150.932
C08774=1107.563,350.149,414.609,-179.155,14.882,150.932
C08775=1107.569,350.397,414.575,-179.152,14.884,150.932
C08776=1107.574,350.644,414.541,-179.148,14.886,150.931
C08777=1107.580,350.892,414.506,-179.146,14.889,150.932
C08778=1107.585,351.139,414.472,-179.142,14.891,150.931
C08779=1107.592,351.387,414.439,-179.139,14.894,150.931
C08780=1107.597,351.635,414.404,-179.136,14.897,150.931
C08781=1107.603,351.882,414.370,-179.133,14.899,150.931
C08782=1107.608,352.130,414.336,-179.129,14.902,150.931
C08783=1107.614,352.377,414.301,-179.126,14.905,150.931
C08784=1107.619,352.625,414.268,-179.123,14.907,150.931
C08785=1107.625,352.872,414.234,-179.120,14.910,150.931
C08786=1107.631,353.120,414.200,-179.117,14.912,150.931
C08787=1107.637,353.368,414.165,-179.114,14.915,150.931
C08788=1107.642,353.615,414.131,-179.111,14.918,150.931
C08789=1107.648,353.862,414.097,-179.107,14.920,150.931
C08790=1107.653,354.110,414.062,-179.105,14.923,150.931
C08791=1107.659,354.357,414.028,-179.101,14.925,150.931
C08792=1107.665,354.606,413.994,-179.098,14.929,150.931
C08793=1107.671,354.854,413.960,-179.095,14.931,150.931
C08794=1107.676,355.101,413.926,-179.092,14.934,150.931
C08795=1107.682,355.348,413.891,-179.089,14.936,150.931
C08796=1107.687,355.596,413.857,-179.085,14.939,150.931
C08797=1107.693,355.844,413.822,-179.083,14.942,150.931
C08798=1107.702,356.214,413.771,-179.077,14.946,150.931
C08799=1107.710,356.585,413.719,-179.073,14.950,150.931
C08800=1107.718,356.954,413.667,-179.068,14.954,150.931
C08801=1107.727,357.325,413.616,-179.064,14.958,150.931
C08802=1107.732,357.572,413.581,-179.061,14.961,150.931
C08803=1107.739,357.820,413.547,-179.057,14.964,150.931
C08804=1107.744,358.068,413.512,-179.054,14.967,150.931
C08805=1107.750,358.315,413.478,-179.052,14.970,150.931
C08806=1107.755,358.563,413.443,-179.048,14.972,150.931
C08807=1107.762,358.810,413.408,-179.045,14.975,150.931
C08808=1107.767,359.058,413.373,-179.042,14.978,150.931
C08809=1107.773,359.305,413.339,-179.039,14.981,150.931
C08810=1107.778,359.553,413.305,-179.036,14.984,150.931
C08811=1107.784,359.800,413.269,-179.033,14.987,150.931
C08812=1107.790,360.048,413.235,-179.030,14.990,150.931
C08813=1107.795,360.295,413.200,-179.027,14.992,150.931
C08814=1107.801,360.543,413.166,-179.024,14.996,150.931
C08815=1107.807,360.790,413.131,-179.021,14.999,150.931
C08816=1107.812,361.038,413.096,-179.018,15.001,150.931
C08817=1107.818,361.285,413.062,-179.015,15.004,150.931
C08818=1107.824,361.533,413.026,-179.011,15.008,150.931
C08819=1107.829,361.780,412.991,-179.009,15.011,150.931
C08820=1107.835,362.028,412.957,-179.006,15.014,150.932
C08821=1107.841,362.275,412.922,-179.003,15.016,150.932
C08822=1107.846,362.523,412.887,-178.999,15.020,150.932
C08823=1107.852,362.769,412.852,-178.997,15.023,150.932
C08824=1107.858,363.018,412.817,-178.994,15.026,150.932
C08825=1107.863,363.265,412.782,-178.991,15.028,150.932
C08826=1107.868,363.512,412.747,-178.987,15.032,150.932
C08827=1107.875,363.760,412.712,-178.985,15.035,150.932
C08828=1107.880,364.007,412.677,-178.982,15.038,150.932
C08829=1107.886,364.254,412.642,-178.979,15.041,150.932
C08830=1107.891,364.503,412.607,-178.976,15.044,150.933
C08831=1107.898,364.749,412.572,-178.973,15.047,150.933
C08832=1107.903,364.997,412.538,-178.970,15.050,150.933
C08833=1107.909,365.244,412.502,-178.967,15.054,150.933
C08834=1107.914,365.492,412.467,-178.964,15.057,150.933
C08835=1107.920,365.740,412.432,-178.961,15.060,150.933
C08836=1107.926,365.986,412.397,-178.959,15.063,150.933
C08837=1107.931,366.234,412.362,-178.955,15.066,150.933
C08838=1107.937,366.482,412.326,-178.952,15.069,150.934
C08839=1107.943,366.729,412.291,-178.950,15.073,150.934
C08840=1107.948,366.977,412.256,-178.946,15.076,150.934
C08841=1107.954,367.224,412.221,-178.944,15.079,150.934
C08842=1107.959,367.471,412.185,-178.941,15.082,150.934
C08843=1107.965,367.719,412.150,-178.937,15.086,150.934
C08844=1107.970,367.966,412.115,-178.935,15.089,150.935
C08845=1107.976,368.213,412.080,-178.932,15.092,150.935
C08846=1107.982,368.461,412.044,-178.929,15.096,150.935
C08847=1107.987,368.708,412.009,-178.926,15.099,150.935
C08848=1107.993,368.956,411.973,-178.923,15.103,150.936
C08849=1107.998,369.203,411.938,-178.920,15.106,150.936
C08850=1108.008,369.588,411.883,-178.916,15.111,150.936
C08851=1108.016,369.973,411.828,-178.912,15.116,150.936
C08852=1108.026,370.358,411.773,-178.907,15.121,150.937
C08853=1108.034,370.744,411.718,-178.902,15.127,150.937
C08854=1108.040,370.991,411.682,-178.900,15.130,150.937
C08855=1108.046,371.238,411.647,-178.897,15.134,150.937
C08856=1108.051,371.485,411.611,-178.894,15.137,150.938
C08857=1108.057,371.733,411.575,-178.891,15.141,150.938
C08858=1108.063,371.980,411.540,-178.888,15.144,150.938
C08859=1108.069,372.228,411.504,-178.886,15.147,150.939
C08860=1108.073,372.475,411.468,-178.883,15.151,150.939
C08861=1108.080,372.723,411.433,-178.880,15.154,150.939
C08862=1108.085,372.970,411.397,-178.877,15.158,150.939
C08863=1108.091,373.217,411.362,-178.874,15.162,150.940
C08864=1108.096,373.464,411.326,-178.871,15.166,150.940
C08865=1108.102,373.712,411.290,-178.869,15.169,150.940
C08866=1108.108,373.959,411.255,-178.866,15.172,150.940
C08867=1108.114,374.207,411.219,-178.863,15.176,150.941
C08868=1108.120,374.453,411.183,-178.860,15.179,150.941
C08869=1108.125,374.701,411.147,-178.857,15.183,150.941
C08870=1108.130,374.948,411.112,-178.855,15.187,150.942
C08871=1108.136,375.196,411.076,-178.852,15.191,150.942
C08872=1108.142,375.443,411.041,-178.849,15.194,150.942
C08873=1108.147,375.691,411.004,-178.846,15.198,150.943
C08874=1108.153,375.937,410.968,-178.844,15.202,150.943
C08875=1108.159,376.185,410.932,-178.841,15.206,150.943
C08876=1108.164,376.432,410.897,-178.838,15.209,150.944
C08877=1108.170,376.680,410.861,-178.836,15.213,150.944
C08878=1108.176,376.927,410.824,-178.833,15.216,150.944
C08879=1108.181,377.174,410.789,-178.830,15.221,150.945
C08880=1108.187,377.422,410.753,-178.828,15.224,150.945
C08881=1108.192,377.668,410.716,-178.825,15.228,150.945
C08882=1108.198,377.916,410.681,-178.822,15.232,150.946
C08883=1108.203,378.163,410.645,-178.819,15.236,150.946
C08884=1108.209,378.410,410.608,-178.817,15.239,150.946
C08885=1108.215,378.658,410.573,-178.814,15.243,150.947
C08886=1108.220,378.905,410.537,-178.812,15.247,150.947
C08887=1108.226,379.152,410.500,-178.809,15.251,150.948
C08888=1108.232,379.399,410.465,-178.806,15.255,150.948
C08889=1108.238,379.646,410.428,-178.803,15.259,150.948
C08890=1108.244,379.894,410.392,-178.800,15.263,150.949
C08891=1108.249,380.140,410.356,-178.798,15.267,150.949
C08892=1108.255,380.388,410.320,-178.795,15.271,150.950
C08893=1108.261,380.635,410.283,-178.793,15.274,150.950
C08894=1108.266,380.883,410.247,-178.790,15.279,150.950
C08895=1108.272,381.130,410.211,-178.788,15.282,150.951
C08896=1108.277,381.377,410.175,-178.785,15.286,150.951
C08897=1108.283,381.624,410.138,-178.782,15.291,150.952
C08898=1108.289,381.871,410.102,-178.780,15.294,150.952
C08899=1108.294,382.118,410.066,-178.777,15.299,150.953
C08900=1108.300,382.365,410.030,-178.774,15.302,150.953
C08901=1108.306,382.613,409.993,-178.771,15.306,150.953
C08902=1108.315,383.025,409.933,-178.767,15.313,150.954
C08903=1108.325,383.437,409.872,-178.763,15.320,150.955
C08904=1108.334,383.848,409.811,-178.759,15.327,150.956
C08905=1108.344,384.260,409.751,-178.754,15.334,150.957
C08906=1108.349,384.507,409.714,-178.752,15.339,150.957
C08907=1108.354,384.755,409.678,-178.749,15.342,150.958
C08908=1108.361,385.002,409.641,-178.747,15.347,150.958
C08909=1108.366,385.249,409.604,-178.744,15.352,150.959
C08910=1108.371,385.496,409.567,-178.742,15.355,150.959
C08911=1108.377,385.743,409.531,-178.739,15.360,150.960
C08912=1108.383,385.991,409.495,-178.736,15.364,150.960
C08913=1108.388,386.238,409.458,-178.735,15.368,150.961
C08914=1108.394,386.485,409.422,-178.732,15.373,150.961
C08915=1108.400,386.732,409.385,-178.729,15.377,150.962
C08916=1108.405,386.979,409.348,-178.727,15.381,150.962
C08917=1108.411,387.226,409.311,-178.724,15.385,150.963
C08918=1108.417,387.473,409.274,-178.722,15.390,150.963
C08919=1108.422,387.720,409.237,-178.719,15.395,150.964
C08920=1108.428,387.967,409.201,-178.717,15.398,150.965
C08921=1108.434,388.214,409.164,-178.714,15.403,150.965
C08922=1108.439,388.462,409.127,-178.712,15.408,150.966
C08923=1108.445,388.709,409.090,-178.709,15.412,150.966
C08924=1108.450,388.955,409.054,-178.707,15.416,150.967
C08925=1108.456,389.203,409.017,-178.705,15.421,150.968
C08926=1108.462,389.450,408.980,-178.702,15.426,150.968
C08927=1108.467,389.697,408.943,-178.699,15.430,150.969
C08928=1108.474,389.944,408.907,-178.697,15.434,150.969
C08929=1108.479,390.192,408.869,-178.695,15.439,150.970
C08930=1108.484,390.438,408.833,-178.692,15.444,150.971
C08931=1108.490,390.686,408.796,-178.689,15.448,150.971
C08932=1108.495,390.933,408.759,-178.687,15.453,150.972
C08933=1108.502,391.180,408.722,-178.685,15.457,150.972
C08934=1108.508,391.427,408.685,-178.682,15.462,150.973
C08935=1108.513,391.674,408.647,-178.680,15.467,150.974
C08936=1108.519,391.922,408.610,-178.677,15.471,150.974
C08937=1108.524,392.168,408.574,-178.675,15.476,150.975
C08938=1108.530,392.415,408.537,-178.673,15.480,150.976
C08939=1108.536,392.662,408.500,-178.671,15.485,150.976
C08940=1108.542,392.910,408.463,-178.668,15.490,150.977
C08941=1108.547,393.157,408.425,-178.666,15.495,150.978
C08942=1108.553,393.404,408.388,-178.663,15.499,150.978
C08943=1108.559,393.651,408.351,-178.662,15.504,150.979
C08944=1108.564,393.898,408.314,-178.659,15.509,150.980
C08945=1108.570,394.146,408.277,-178.657,15.514,150.981
C08946=1108.575,394.392,408.239,-178.655,15.518,150.981
C08947=1108.581,394.639,408.202,-178.652,15.523,150.982
C08948=1108.586,394.886,408.165,-178.650,15.528,150.983
C08949=1108.592,395.133,408.127,-178.647,15.533,150.984
C08950=1108.598,395.381,408.090,-178.645,15.538,150.984
C08951=1108.604,395.628,408.053,-178.643,15.543,150.985
C08952=1108.609,395.875,408.016,-178.641,15.548,150.986
C08953=1108.614,396.122,407.978,-178.639,15.552,150.986
C08954=1108.620,396.334,407.946,-178.637,15.557,150.987
C08955=1108.625,396.546,407.914,-178.635,15.562,150.988
C08956=1108.629,396.757,407.882,-178.633,15.566,150.988
C08957=1108.634,396.970,407.850,-178.631,15.570,150.989
C08958=1108.639,397.181,407.817,-178.629,15.574,150.990
C08959=1108.644,397.394,407.786,-178.627,15.579,150.991
C08960=1108.648,397.605,407.753,-178.625,15.583,150.991
C08961=1108.653,397.817,407.721,-178.623,15.587,150.992
C08962=1108.659,398.064,407.683,-178.621,15.592,150.993
C08963=1108.665,398.312,407.646,-178.619,15.597,150.994
C08964=1108.670,398.559,407.608,-178.617,15.603,150.994
C08965=1108.676,398.806,407.571,-178.614,15.608,150.995
C08966=1108.682,399.053,407.533,-178.612,15.613,150.996
C08967=1108.687,399.299,407.496,-178.610,15.618,150.997
C08968=1108.693,399.547,407.459,-178.608,15.623,150.998
C08969=1108.698,399.794,407.420,-178.606,15.629,150.999
C08970=1108.704,400.041,407.382,-178.604,15.634,151.000
C08971=1108.710,400.288,407.345,-178.602,15.639,151.000
C08972=1108.715,400.535,407.307,-178.600,15.644,151.001
C08973=1108.721,400.782,407.269,-178.597,15.649,151.002
C08974=1108.726,401.029,407.232,-178.595,15.655,151.003
C08975=1108.732,401.276,407.194,-178.593,15.660,151.004
C08976=1108.738,401.524,407.156,-178.591,15.666,151.005
C08977=1108.744,401.771,407.119,-178.589,15.671,151.006
C08978=1108.749,402.018,407.080,-178.587,15.676,151.007
C08979=1108.755,402.265,407.043,-178.585,15.682,151.008
C08980=1108.761,402.512,407.005,-178.583,15.687,151.009
C08981=1108.766,402.759,406.967,-178.581,15.692,151.009
C08982=1108.771,403.006,406.929,-178.578,15.699,151.011
C08983=1108.777,403.253,406.892,-178.576,15.704,151.011
C08984=1108.782,403.500,406.853,-178.574,15.709,151.012
C08985=1108.788,403.747,406.816,-178.572,15.715,151.013
C08986=1108.794,403.994,406.777,-178.570,15.720,151.014
C08987=1108.800,404.241,406.739,-178.568,15.726,151.015
C08988=1108.806,404.488,406.701,-178.566,15.731,151.016
C08989=1108.811,404.735,406.663,-178.564,15.737,151.017
C08990=1108.817,404.982,406.625,-178.562,15.743,151.018
C08991=1108.822,405.229,406.588,-178.560,15.749,151.019
C08992=1108.828,405.476,406.550,-178.558,15.754,151.020
C08993=1108.834,405.724,406.511,-178.556,15.760,151.021
C08994=1108.839,405.971,406.473,-178.554,15.765,151.022
C08995=1108.845,406.218,406.435,-178.552,15.772,151.023
C08996=1108.851,406.464,406.397,-178.550,15.777,151.024
C08997=1108.856,406.711,406.358,-178.548,15.783,151.025
C08998=1108.861,406.958,406.320,-178.547,15.789,151.027
C08999=1108.868,407.205,406.282,-178.545,15.794,151.028
C09000=1108.873,407.452,406.243,-178.542,15.801,151.029
C09001=1108.879,407.699,406.206,-178.540,15.806,151.030
C09002=1108.884,407.946,406.167,-178.539,15.812,151.031
C09003=1108.889,408.193,406.129,-178.536,15.818,151.032
C09004=1108.896,408.441,406.091,-178.534,15.824,151.033
C09005=1108.901,408.688,406.052,-178.533,15.830,151.034
C09006=1108.906,408.934,406.013,-178.531,15.836,151.035
C09007=1108.912,409.181,405.976,-178.529,15.842,151.036
C09008=1108.917,409.428,405.937,-178.527,15.848,151.038
C09009=1108.923,409.676,405.899,-178.525,15.854,151.039
C09010=1108.928,409.886,405.865,-178.524,15.860,151.040
C09011=1108.933,410.099,405.832,-178.522,15.865,151.041
C09012=1108.937,410.310,405.800,-178.520,15.870,151.042
C09013=1108.942,410.522,405.767,-178.519,15.876,151.043
C09014=1108.948,410.733,405.734,-178.517,15.881,151.044
C09015=1108.952,410.945,405.701,-178.516,15.886,151.045
C09016=1108.957,411.157,405.668,-178.514,15.891,151.046
C09017=1108.962,411.369,405.635,-178.512,15.896,151.047
C09018=1108.967,411.615,405.596,-178.510,15.903,151.048
C09019=1108.972,411.862,405.557,-178.509,15.909,151.049
C09020=1108.979,412.109,405.519,-178.507,15.915,151.050
C09021=1108.984,412.356,405.480,-178.505,15.922,151.052
C09022=1108.989,412.603,405.442,-178.504,15.928,151.053
C09023=1108.995,412.850,405.403,-178.501,15.935,151.054
C09024=1109.001,413.098,405.364,-178.500,15.941,151.055
C09025=1109.006,413.344,405.325,-178.498,15.948,151.056
C09026=1109.012,413.591,405.287,-178.496,15.954,151.058
C09027=1109.018,413.838,405.248,-178.494,15.960,151.059
C09028=1109.023,414.085,405.210,-178.493,15.967,151.060
C09029=1109.029,414.331,405.170,-178.490,15.973,151.062
C09030=1109.035,414.579,405.132,-178.489,15.979,151.063
C09031=1109.040,414.826,405.093,-178.487,15.987,151.064
C09032=1109.046,415.072,405.054,-178.485,15.993,151.065
C09033=1109.052,415.319,405.016,-178.484,16.000,151.067
C09034=1109.057,415.566,404.976,-178.482,16.006,151.068
C09035=1109.063,415.813,404.938,-178.480,16.013,151.069
C09036=1109.069,416.060,404.899,-178.479,16.019,151.071
C09037=1109.074,416.306,404.860,-178.477,16.026,151.072
C09038=1109.080,416.554,404.821,-178.475,16.032,151.073
C09039=1109.085,416.801,404.782,-178.473,16.039,151.075
C09040=1109.091,417.047,404.743,-178.471,16.046,151.076
C09041=1109.097,417.294,404.703,-178.470,16.053,151.078
C09042=1109.102,417.541,404.665,-178.468,16.060,151.079
C09043=1109.108,417.788,404.626,-178.467,16.066,151.080
C09044=1109.114,418.035,404.586,-178.465,16.073,151.082
C09045=1109.119,418.281,404.547,-178.463,16.080,151.083
C09046=1109.124,418.528,404.509,-178.462,16.087,151.084
C09047=1109.130,418.775,404.470,-178.460,16.094,151.086
C09048=1109.136,419.022,404.431,-178.458,16.101,151.087
C09049=1109.141,419.269,404.391,-178.457,16.108,151.089
C09050=1109.147,419.516,404.351,-178.455,16.115,151.090
C09051=1109.152,419.762,404.312,-178.454,16.123,151.092
C09052=1109.158,420.009,404.273,-178.453,16.129,151.093
C09053=1109.164,420.256,404.234,-178.451,16.137,151.095
C09054=1109.169,420.504,404.195,-178.449,16.144,151.096
C09055=1109.175,420.750,404.156,-178.447,16.151,151.098
C09056=1109.181,420.997,404.117,-178.446,16.158,151.099
C09057=1109.186,421.244,404.077,-178.445,16.165,151.101
C09058=1109.191,421.490,404.038,-178.443,16.173,151.102
C09059=1109.197,421.737,403.999,-178.441,16.180,151.104
